C01786=1124.432,191.040,-64.237,-179.146,9.228,149.571
C01787=1124.436,190.791,-64.212,-179.148,9.226,149.571
C01788=1124.441,190.542,-64.188,-179.151,9.223,149.571
C01789=1124.446,190.294,-64.164,-179.153,9.220,149.570
C01790=1124.450,190.046,-64.139,-179.155,9.217,149.570
C01791=1124.455,189.796,-64.114,-179.157,9.214,149.570
C01792=1124.459,189.548,-64.090,-179.159,9.211,149.570
C01793=1124.464,189.299,-64.067,-179.161,9.209,149.570
C01794=1124.469,189.050,-64.042,-179.164,9.206,149.570
C01795=1124.473,188.801,-64.018,-179.166,9.204,149.570
C01796=1124.477,188.553,-63.994,-179.168,9.200,149.570
C01797=1124.482,188.304,-63.969,-179.170,9.198,149.570
C01798=1124.487,188.055,-63.946,-179.172,9.195,149.570
C01799=1124.491,187.806,-63.922,-179.175,9.192,149.570
C01800=1124.495,187.557,-63.897,-179.177,9.190,149.570
C01801=1124.500,187.309,-63.873,-179.179,9.186,149.570
C01802=1124.505,187.059,-63.849,-179.182,9.184,149.570
C01803=1124.509,186.811,-63.825,-179.184,9.181,149.570
C01804=1124.514,186.563,-63.801,-179.187,9.178,149.570
C01805=1124.519,186.313,-63.777,-179.189,9.175,149.570
C01806=1124.523,186.064,-63.753,-179.192,9.172,149.570
C01807=1124.528,185.850,-63.732,-179.194,9.170,149.570
C01808=1124.530,185.637,-63.711,-179.196,9.167,149.570
C01809=1124.534,185.422,-63.691,-179.198,9.164,149.570
C01810=1124.539,185.208,-63.670,-179.200,9.162,149.570
C01811=1124.543,184.994,-63.649,-179.202,9.160,149.570
C01812=1124.547,184.780,-63.630,-179.205,9.157,149.570
C01813=1124.550,184.566,-63.608,-179.207,9.155,149.570
C01814=1124.555,184.352,-63.588,-179.209,9.151,149.570
C01815=1124.559,184.102,-63.564,-179.212,9.148,149.570
C01816=1124.563,183.854,-63.540,-179.214,9.145,149.570
C01817=1124.568,183.605,-63.517,-179.217,9.142,149.570
C01818=1124.572,183.357,-63.493,-179.220,9.139,149.570
C01819=1124.577,183.108,-63.468,-179.222,9.136,149.570
C01820=1124.581,182.859,-63.445,-179.225,9.133,149.570
C01821=1124.586,182.611,-63.421,-179.227,9.130,149.570
C01822=1124.591,182.361,-63.397,-179.230,9.127,149.570
C01823=1124.596,182.112,-63.374,-179.233,9.124,149.570
C01824=1124.600,181.864,-63.350,-179.236,9.120,149.570
C01825=1124.604,181.614,-63.326,-179.239,9.117,149.570
C01826=1124.609,181.366,-63.302,-179.241,9.114,149.570
C01827=1124.613,181.117,-63.279,-179.244,9.111,149.570
C01828=1124.618,180.868,-63.254,-179.247,9.107,149.570
C01829=1124.623,180.619,-63.231,-179.250,9.104,149.570
C01830=1124.627,180.370,-63.208,-179.252,9.101,149.570
C01831=1124.632,180.122,-63.184,-179.256,9.098,149.570
C01832=1124.636,179.873,-63.160,-179.258,9.095,149.570
C01833=1124.641,179.624,-63.137,-179.261,9.091,149.570
C01834=1124.645,179.375,-63.113,-179.264,9.088,149.570
C01835=1124.650,179.126,-63.089,-179.267,9.085,149.570
C01836=1124.654,178.878,-63.067,-179.269,9.081,149.570
C01837=1124.659,178.629,-63.043,-179.271,9.079,149.570
C01838=1124.663,178.380,-63.019,-179.273,9.076,149.569
C01839=1124.668,178.131,-62.996,-179.276,9.073,149.569
C01840=1124.673,177.882,-62.973,-179.277,9.070,149.569
C01841=1124.677,177.633,-62.949,-179.280,9.067,149.569
C01842=1124.682,177.385,-62.925,-179.282,9.064,149.569
C01843=1124.686,177.136,-62.902,-179.284,9.061,149.569
C01844=1124.691,176.887,-62.878,-179.286,9.058,149.569
C01845=1124.696,176.638,-62.855,-179.288,9.055,149.569
C01846=1124.700,176.389,-62.832,-179.290,9.052,149.569
C01847=1124.704,176.140,-62.809,-179.293,9.049,149.568
C01848=1124.709,175.891,-62.785,-179.294,9.047,149.568
C01849=1124.714,175.642,-62.762,-179.297,9.043,149.568
C01850=1124.718,175.393,-62.738,-179.299,9.040,149.568
C01851=1124.723,175.144,-62.715,-179.301,9.038,149.568
C01852=1124.727,174.896,-62.692,-179.304,9.035,149.568
C01853=1124.732,174.647,-62.669,-179.306,9.031,149.568
C01854=1124.737,174.398,-62.646,-179.308,9.028,149.568
C01855=1124.742,174.149,-62.622,-179.310,9.026,149.568
C01856=1124.746,173.900,-62.599,-179.313,9.022,149.568
C01857=1124.750,173.652,-62.576,-179.315,9.019,149.567
C01858=1124.755,173.402,-62.553,-179.317,9.017,149.567
C01859=1124.760,173.153,-62.529,-179.319,9.014,149.567
C01860=1124.764,172.904,-62.506,-179.321,9.010,149.567
C01861=1124.768,172.656,-62.483,-179.324,9.007,149.567
C01862=1124.773,172.407,-62.460,-179.326,9.005,149.567
C01863=1124.778,172.193,-62.440,-179.328,9.002,149.567
C01864=1124.781,171.979,-62.420,-179.330,8.999,149.567
C01865=1124.785,171.764,-62.400,-179.331,8.997,149.567
C01866=1124.789,171.550,-62.380,-179.333,8.994,149.567
C01867=1124.793,171.336,-62.361,-179.335,8.992,149.567
C01868=1124.797,171.122,-62.341,-179.337,8.988,149.566
C01869=1124.801,170.908,-62.320,-179.339,8.986,149.566
C01870=1124.805,170.694,-62.301,-179.341,8.984,149.566
C01871=1124.810,170.445,-62.278,-179.344,8.981,149.566
C01872=1124.814,170.196,-62.255,-179.346,8.977,149.566
C01873=1124.819,169.947,-62.232,-179.348,8.974,149.566
C01874=1124.823,169.698,-62.208,-179.350,8.972,149.566
C01875=1124.827,169.449,-62.186,-179.353,8.969,149.566
C01876=1124.833,169.200,-62.163,-179.355,8.965,149.566
C01877=1124.837,168.951,-62.140,-179.357,8.962,149.566
C01878=1124.841,168.703,-62.117,-179.360,8.959,149.566
C01879=1124.846,168.454,-62.094,-179.362,8.955,149.565
C01880=1124.851,168.204,-62.071,-179.364,8.953,149.565
C01881=1124.856,167.956,-62.049,-179.366,8.950,149.565
C01882=1124.860,167.707,-62.025,-179.369,8.947,149.565
C01883=1124.864,167.458,-62.003,-179.371,8.943,149.565
C01884=1124.869,167.209,-61.980,-179.373,8.940,149.565
C01885=1124.875,166.960,-61.957,-179.376,8.937,149.565
C01886=1124.879,166.712,-61.934,-179.378,8.934,149.565
C01887=1124.884,166.462,-61.912,-179.381,8.931,149.565
C01888=1124.888,166.213,-61.889,-179.383,8.927,149.565
C01889=1124.893,165.965,-61.866,-179.385,8.925,149.565
C01890=1124.897,165.715,-61.844,-179.387,8.922,149.564
C01891=1124.902,165.466,-61.820,-179.390,8.919,149.564
C01892=1124.906,165.218,-61.798,-179.392,8.915,149.564
C01893=1124.911,164.969,-61.775,-179.395,8.912,149.564
C01894=1124.915,164.720,-61.753,-179.397,8.909,149.564
C01895=1124.920,164.470,-61.730,-179.399,8.906,149.564
C01896=1124.925,164.222,-61.708,-179.402,8.903,149.564
C01897=1124.930,163.973,-61.685,-179.404,8.899,149.564
C01898=1124.934,163.724,-61.662,-179.406,8.896,149.564
C01899=1124.939,163.475,-61.639,-179.409,8.893,149.564
C01900=1124.944,163.226,-61.617,-179.411,8.889,149.563
C01901=1124.947,162.978,-61.594,-179.414,8.886,149.563
C01902=1124.952,162.728,-61.572,-179.416,8.883,149.563
C01903=1124.957,162.480,-61.549,-179.419,8.880,149.563
C01904=1124.962,162.230,-61.527,-179.421,8.877,149.563
C01905=1124.966,161.981,-61.505,-179.423,8.873,149.563
C01906=1124.971,161.733,-61.482,-179.426,8.870,149.563
C01907=1124.976,161.483,-61.460,-179.428,8.867,149.563
C01908=1124.980,161.235,-61.437,-179.430,8.864,149.563
C01909=1124.985,160.986,-61.415,-179.433,8.861,149.563
C01910=1124.989,160.737,-61.392,-179.435,8.857,149.563
C01911=1124.994,160.488,-61.370,-179.438,8.853,149.563
C01912=1124.999,160.239,-61.348,-179.441,8.850,149.562
C01913=1125.003,159.990,-61.325,-179.443,8.847,149.562
C01914=1125.008,159.741,-61.303,-179.445,8.844,149.562
C01915=1125.012,159.492,-61.281,-179.447,8.840,149.562
C01916=1125.017,159.243,-61.258,-179.450,8.837,149.562
C01917=1125.022,158.994,-61.236,-179.452,8.834,149.562
C01918=1125.026,158.745,-61.214,-179.454,8.830,149.562
C01919=1125.030,158.531,-61.195,-179.457,8.827,149.562
C01920=1125.034,158.316,-61.176,-179.459,8.824,149.562
C01921=1125.038,158.102,-61.157,-179.461,8.821,149.561
C01922=1125.043,157.888,-61.138,-179.463,8.818,149.561
C01923=1125.047,157.674,-61.118,-179.465,8.816,149.561
C01924=1125.050,157.459,-61.099,-179.467,8.813,149.561
C01925=1125.054,157.245,-61.080,-179.470,8.809,149.561
C01926=1125.058,157.031,-61.061,-179.471,8.807,149.561
C01927=1125.063,156.782,-61.039,-179.474,8.804,149.561
C01928=1125.068,156.532,-61.017,-179.477,8.800,149.561
C01929=1125.073,156.284,-60.994,-179.479,8.796,149.561
C01930=1125.077,156.035,-60.972,-179.482,8.793,149.561
C01931=1125.082,155.786,-60.950,-179.484,8.790,149.560
C01932=1125.086,155.537,-60.928,-179.487,8.786,149.560
C01933=1125.090,155.288,-60.906,-179.489,8.782,149.560
C01934=1125.096,155.039,-60.884,-179.491,8.779,149.560
C01935=1125.101,154.790,-60.862,-179.494,8.776,149.560
C01936=1125.105,154.541,-60.840,-179.497,8.772,149.560
C01937=1125.110,154.292,-60.819,-179.499,8.768,149.559
C01938=1125.114,154.043,-60.797,-179.501,8.765,149.559
C01939=1125.119,153.794,-60.775,-179.504,8.761,149.559
C01940=1125.123,153.545,-60.753,-179.507,8.758,149.559
C01941=1125.128,153.296,-60.731,-179.509,8.754,149.559
C01942=1125.133,153.047,-60.709,-179.512,8.750,149.559
C01943=1125.138,152.798,-60.687,-179.514,8.747,149.559
C01944=1125.142,152.549,-60.665,-179.516,8.744,149.559
C01945=1125.147,152.300,-60.643,-179.519,8.740,149.558
C01946=1125.152,152.051,-60.621,-179.521,8.736,149.558
C01947=1125.156,151.802,-60.599,-179.524,8.732,149.558
C01948=1125.161,151.553,-60.578,-179.526,8.729,149.558
C01949=1125.166,151.304,-60.556,-179.529,8.726,149.558
C01950=1125.170,151.055,-60.534,-179.532,8.721,149.558
C01951=1125.175,150.805,-60.513,-179.534,8.718,149.557
C01952=1125.180,150.557,-60.491,-179.537,8.714,149.557
C01953=1125.185,150.308,-60.469,-179.539,8.711,149.557
C01954=1125.189,150.059,-60.447,-179.542,8.707,149.557
C01955=1125.194,149.810,-60.426,-179.544,8.703,149.557
C01956=1125.199,149.561,-60.405,-179.547,8.699,149.557
C01957=1125.203,149.311,-60.383,-179.549,8.696,149.557
C01958=1125.208,149.063,-60.361,-179.552,8.692,149.556
C01959=1125.213,148.814,-60.339,-179.554,8.688,149.556
C01960=1125.217,148.565,-60.318,-179.557,8.684,149.556
C01961=1125.222,148.316,-60.297,-179.559,8.681,149.556
C01962=1125.227,148.067,-60.275,-179.562,8.676,149.556
C01963=1125.231,147.818,-60.253,-179.564,8.673,149.555
C01964=1125.236,147.569,-60.232,-179.567,8.669,149.555
C01965=1125.241,147.320,-60.210,-179.569,8.666,149.555
C01966=1125.246,147.070,-60.189,-179.572,8.661,149.555
C01967=1125.250,146.821,-60.167,-179.575,8.657,149.555
C01968=1125.255,146.573,-60.146,-179.577,8.654,149.554
C01969=1125.259,146.323,-60.125,-179.580,8.650,149.554
C01970=1125.264,146.074,-60.103,-179.582,8.646,149.554
C01971=1125.269,145.825,-60.082,-179.585,8.642,149.554
C01972=1125.274,145.577,-60.061,-179.588,8.638,149.554
C01973=1125.278,145.328,-60.039,-179.590,8.634,149.554
C01974=1125.283,145.078,-60.018,-179.592,8.630,149.553
C01975=1125.287,144.863,-60.000,-179.594,8.627,149.553
C01976=1125.290,144.650,-59.981,-179.595,8.624,149.553
C01977=1125.295,144.435,-59.963,-179.596,8.621,149.552
C01978=1125.299,144.220,-59.945,-179.598,8.619,149.552
C01979=1125.303,144.007,-59.926,-179.599,8.616,149.552
C01980=1125.308,143.792,-59.908,-179.600,8.613,149.552
C01981=1125.311,143.577,-59.890,-179.601,8.610,149.551
C01982=1125.315,143.363,-59.871,-179.603,8.607,149.551
C01983=1125.320,143.114,-59.851,-179.604,8.603,149.550
C01984=1125.324,142.864,-59.829,-179.606,8.600,149.550
C01985=1125.329,142.616,-59.808,-179.607,8.597,149.550
C01986=1125.334,142.367,-59.787,-179.609,8.594,149.550
C01987=1125.339,142.118,-59.766,-179.611,8.590,149.549
C01988=1125.344,141.869,-59.745,-179.612,8.587,149.549
C01989=1125.348,141.619,-59.723,-179.614,8.583,149.548
C01990=1125.352,141.371,-59.702,-179.615,8.580,149.548
C01991=1125.358,141.121,-59.681,-179.617,8.577,149.548
C01992=1125.362,140.873,-59.660,-179.618,8.574,149.547
C01993=1125.367,140.624,-59.639,-179.620,8.570,149.547
C01994=1125.371,140.374,-59.618,-179.621,8.567,149.547
C01995=1125.376,140.125,-59.597,-179.623,8.564,149.546
C01996=1125.381,139.876,-59.576,-179.624,8.561,149.546
C01997=1125.386,139.627,-59.555,-179.626,8.557,149.546
C01998=1125.390,139.378,-59.535,-179.627,8.554,149.545
C01999=1125.395,139.129,-59.513,-179.629,8.551,149.545
C02000=1125.399,138.880,-59.492,-179.630,8.547,149.545
C02001=1125.404,138.630,-59.471,-179.632,8.544,149.544
C02002=1125.409,138.381,-59.450,-179.634,8.541,149.544
C02003=1125.414,138.133,-59.429,-179.635,8.537,149.544
C02004=1125.419,137.884,-59.408,-179.637,8.535,149.544
C02005=1125.423,137.635,-59.388,-179.638,8.531,149.543
C02006=1125.428,137.385,-59.367,-179.640,8.527,149.543
C02007=1125.432,137.137,-59.346,-179.641,8.524,149.543
C02008=1125.437,136.887,-59.324,-179.643,8.521,149.542
C02009=1125.442,136.638,-59.303,-179.644,8.518,149.542
C02010=1125.447,136.389,-59.283,-179.647,8.514,149.542
C02011=1125.452,136.140,-59.262,-179.648,8.511,149.541
C02012=1125.456,135.891,-59.242,-179.650,8.508,149.541
C02013=1125.461,135.642,-59.220,-179.651,8.505,149.541
C02014=1125.466,135.393,-59.200,-179.653,8.501,149.541
C02015=1125.471,135.144,-59.179,-179.655,8.497,149.540
C02016=1125.475,134.895,-59.158,-179.656,8.495,149.540
C02017=1125.480,134.646,-59.137,-179.658,8.491,149.539
C02018=1125.485,134.397,-59.117,-179.659,8.488,149.539
C02019=1125.489,134.147,-59.096,-179.661,8.485,149.539
C02020=1125.494,133.898,-59.075,-179.662,8.482,149.539
C02021=1125.498,133.649,-59.055,-179.664,8.478,149.538
C02022=1125.503,133.400,-59.034,-179.667,8.475,149.538
C02023=1125.508,133.151,-59.014,-179.668,8.471,149.538
C02024=1125.513,132.901,-58.993,-179.670,8.468,149.537
C02025=1125.517,132.652,-58.972,-179.671,8.465,149.537
C02026=1125.523,132.403,-58.951,-179.673,8.461,149.537
C02027=1125.527,132.154,-58.931,-179.675,8.458,149.537
C02028=1125.532,131.905,-58.911,-179.676,8.455,149.536
C02029=1125.537,131.656,-58.890,-179.678,8.451,149.536
C02030=1125.541,131.407,-58.869,-179.679,8.449,149.536
C02031=1125.546,131.192,-58.851,-179.681,8.445,149.535
C02032=1125.550,130.978,-58.833,-179.683,8.442,149.535
C02033=1125.553,130.764,-58.816,-179.684,8.440,149.535
C02034=1125.557,130.549,-58.799,-179.686,8.437,149.535
C02035=1125.562,130.335,-58.781,-179.687,8.434,149.534
C02036=1125.566,130.120,-58.763,-179.688,8.431,149.534
C02037=1125.570,129.906,-58.745,-179.690,8.428,149.534
C02038=1125.574,129.691,-58.728,-179.691,8.426,149.534
C02039=1125.579,129.442,-58.707,-179.693,8.422,149.533
C02040=1125.584,129.193,-58.687,-179.695,8.419,149.533
C02041=1125.588,128.944,-58.667,-179.696,8.416,149.533
C02042=1125.593,128.695,-58.646,-179.698,8.412,149.533
C02043=1125.598,128.446,-58.625,-179.700,8.409,149.532
C02044=1125.603,128.196,-58.606,-179.702,8.406,149.532
C02045=1125.608,127.947,-58.585,-179.703,8.402,149.532
C02046=1125.612,127.698,-58.564,-179.705,8.399,149.531
C02047=1125.617,127.449,-58.544,-179.707,8.396,149.531
C02048=1125.621,127.200,-58.524,-179.709,8.392,149.531
C02049=1125.627,126.950,-58.503,-179.711,8.389,149.531
C02050=1125.631,126.701,-58.483,-179.712,8.386,149.530
C02051=1125.635,126.452,-58.463,-179.714,8.382,149.530
C02052=1125.640,126.204,-58.442,-179.716,8.379,149.530
C02053=1125.645,125.954,-58.422,-179.717,8.376,149.529
C02054=1125.650,125.705,-58.402,-179.719,8.372,149.529
C02055=1125.655,125.456,-58.382,-179.721,8.369,149.529
C02056=1125.660,125.207,-58.362,-179.723,8.366,149.529
C02057=1125.664,124.958,-58.342,-179.724,8.362,149.528
C02058=1125.669,124.709,-58.321,-179.726,8.359,149.528
C02059=1125.674,124.459,-58.301,-179.728,8.355,149.528
C02060=1125.678,124.210,-58.281,-179.730,8.352,149.528
C02061=1125.683,123.961,-58.260,-179.732,8.349,149.527
C02062=1125.688,123.712,-58.241,-179.734,8.345,149.527
C02063=1125.693,123.463,-58.221,-179.735,8.342,149.527
C02064=1125.697,123.214,-58.201,-179.737,8.339,149.527
C02065=1125.703,122.965,-58.180,-179.739,8.335,149.526
C02066=1125.707,122.716,-58.160,-179.741,8.331,149.526
C02067=1125.712,122.466,-58.140,-179.742,8.329,149.526
C02068=1125.716,122.217,-58.119,-179.744,8.325,149.525
C02069=1125.722,121.968,-58.100,-179.746,8.322,149.525
C02070=1125.726,121.719,-58.080,-179.748,8.318,149.525
C02071=1125.731,121.470,-58.060,-179.749,8.315,149.525
C02072=1125.735,121.221,-58.040,-179.752,8.312,149.524
C02073=1125.740,120.971,-58.020,-179.754,8.308,149.524
C02074=1125.744,120.722,-58.000,-179.756,8.305,149.524
C02075=1125.750,120.473,-57.980,-179.757,8.302,149.524
C02076=1125.755,120.224,-57.960,-179.759,8.298,149.523
C02077=1125.760,119.975,-57.940,-179.761,8.295,149.523
C02078=1125.764,119.726,-57.919,-179.763,8.291,149.523
C02079=1125.769,119.476,-57.900,-179.765,8.288,149.523
C02080=1125.774,119.227,-57.881,-179.766,8.285,149.522
C02081=1125.779,118.978,-57.860,-179.768,8.281,149.522
C02082=1125.783,118.729,-57.841,-179.770,8.277,149.522
C02083=1125.788,118.480,-57.820,-179.772,8.274,149.522
C02084=1125.793,118.231,-57.801,-179.774,8.270,149.521
C02085=1125.798,117.981,-57.781,-179.776,8.268,149.521
C02086=1125.802,117.732,-57.761,-179.777,8.264,149.521
C02087=1125.807,117.518,-57.744,-179.779,8.260,149.520
C02088=1125.810,117.303,-57.728,-179.781,8.258,149.520
C02089=1125.815,117.089,-57.711,-179.782,8.255,149.520
C02090=1125.818,116.874,-57.693,-179.784,8.251,149.520
C02091=1125.823,116.660,-57.677,-179.786,8.249,149.520
C02092=1125.827,116.445,-57.659,-179.787,8.246,149.519
C02093=1125.831,116.230,-57.643,-179.789,8.243,149.519
C02094=1125.835,116.016,-57.625,-179.791,8.240,149.519
C02095=1125.840,115.766,-57.605,-179.793,8.236,149.519
C02096=1125.845,115.517,-57.586,-179.795,8.233,149.518
C02097=1125.850,115.268,-57.566,-179.796,8.230,149.518
C02098=1125.855,115.018,-57.547,-179.798,8.226,149.518
C02099=1125.859,114.770,-57.527,-179.800,8.223,149.518
C02100=1125.864,114.521,-57.508,-179.802,8.219,149.517
C02101=1125.868,114.271,-57.488,-179.804,8.216,149.517
C02102=1125.874,114.022,-57.469,-179.806,8.212,149.517
C02103=1125.878,113.773,-57.449,-179.808,8.208,149.516
C02104=1125.883,113.523,-57.429,-179.810,8.205,149.516
C02105=1125.888,113.275,-57.409,-179.812,8.201,149.516
C02106=1125.892,113.026,-57.390,-179.813,8.198,149.516
C02107=1125.897,112.776,-57.371,-179.815,8.195,149.515
C02108=1125.902,112.527,-57.351,-179.817,8.191,149.515
C02109=1125.907,112.278,-57.332,-179.819,8.188,149.515
C02110=1125.912,112.029,-57.312,-179.821,8.184,149.515
C02111=1125.917,111.779,-57.293,-179.823,8.180,149.514
C02112=1125.921,111.530,-57.274,-179.825,8.177,149.514
C02113=1125.926,111.281,-57.254,-179.827,8.173,149.514
C02114=1125.931,111.031,-57.235,-179.829,8.170,149.514
C02115=1125.937,110.783,-57.215,-179.831,8.166,149.513
C02116=1125.941,110.533,-57.196,-179.834,8.162,149.513
C02117=1125.945,110.284,-57.177,-179.836,8.159,149.513
C02118=1125.951,110.035,-57.157,-179.838,8.154,149.513
C02119=1125.955,109.785,-57.138,-179.840,8.151,149.512
C02120=1125.960,109.537,-57.119,-179.843,8.147,149.512
C02121=1125.965,109.287,-57.099,-179.846,8.142,149.512
C02122=1125.969,109.038,-57.080,-179.848,8.139,149.512
C02123=1125.974,108.789,-57.061,-179.850,8.134,149.512
C02124=1125.979,108.539,-57.041,-179.853,8.131,149.511
C02125=1125.984,108.291,-57.022,-179.855,8.127,149.511
C02126=1125.988,108.041,-57.003,-179.857,8.123,149.511
C02127=1125.994,107.792,-56.985,-179.860,8.119,149.511
C02128=1125.999,107.542,-56.965,-179.862,8.115,149.511
C02129=1126.003,107.294,-56.946,-179.865,8.111,149.510
C02130=1126.008,107.044,-56.927,-179.867,8.108,149.510
C02131=1126.013,106.796,-56.908,-179.869,8.103,149.510
C02132=1126.018,106.545,-56.889,-179.871,8.099,149.509
C02133=1126.023,106.297,-56.870,-179.874,8.095,149.509
C02134=1126.027,106.047,-56.851,-179.876,8.092,149.509
C02135=1126.032,105.798,-56.831,-179.878,8.088,149.509
C02136=1126.037,105.549,-56.813,-179.880,8.083,149.508
C02137=1126.042,105.300,-56.794,-179.882,8.080,149.508
C02138=1126.046,105.050,-56.775,-179.885,8.076,149.508
C02139=1126.051,104.802,-56.755,-179.887,8.072,149.508
C02140=1126.056,104.552,-56.737,-179.889,8.068,149.507
C02141=1126.061,104.303,-56.718,-179.891,8.064,149.507
C02142=1126.066,104.054,-56.699,-179.893,8.061,149.507
C02143=1126.070,103.839,-56.683,-179.895,8.057,149.506
C02144=1126.074,103.624,-56.666,-179.897,8.053,149.506
C02145=1126.078,103.410,-56.650,-179.899,8.050,149.506
C02146=1126.082,103.194,-56.633,-179.900,8.047,149.506
C02147=1126.086,102.980,-56.617,-179.902,8.043,149.505
C02148=1126.091,102.765,-56.601,-179.904,8.040,149.505
C02149=1126.095,102.551,-56.585,-179.906,8.036,149.505
C02150=1126.099,102.335,-56.569,-179.908,8.033,149.505
C02151=1126.104,102.087,-56.550,-179.910,8.029,149.504
C02152=1126.108,101.838,-56.532,-179.912,8.025,149.504
C02153=1126.113,101.588,-56.513,-179.913,8.021,149.504
C02154=1126.118,101.339,-56.494,-179.916,8.017,149.503
C02155=1126.124,101.090,-56.475,-179.918,8.013,149.503
C02156=1126.128,100.841,-56.456,-179.920,8.010,149.503
C02157=1126.133,100.591,-56.438,-179.922,8.005,149.502
C02158=1126.137,100.342,-56.419,-179.924,8.001,149.502
C02159=1126.142,100.093,-56.401,-179.926,7.998,149.502
C02160=1126.148,99.843,-56.382,-179.928,7.994,149.501
C02161=1126.152,99.594,-56.363,-179.930,7.989,149.501
C02162=1126.157,99.345,-56.345,-179.932,7.985,149.501
C02163=1126.162,99.096,-56.326,-179.934,7.982,149.500
C02164=1126.167,98.846,-56.307,-179.935,7.978,149.500
C02165=1126.171,98.597,-56.289,-179.937,7.973,149.499
C02166=1126.177,98.348,-56.270,-179.940,7.970,149.499
C02167=1126.182,98.099,-56.252,-179.941,7.966,149.499
C02168=1126.186,97.849,-56.234,-179.943,7.962,149.498
C02169=1126.191,97.600,-56.215,-179.945,7.957,149.498
C02170=1126.196,97.351,-56.197,-179.947,7.954,149.498
C02171=1126.201,97.101,-56.178,-179.949,7.950,149.497
C02172=1126.205,96.853,-56.159,-179.950,7.946,149.497
C02173=1126.211,96.603,-56.141,-179.952,7.942,149.496
C02174=1126.216,96.354,-56.123,-179.953,7.938,149.496
C02175=1126.220,96.104,-56.105,-179.956,7.934,149.496
C02176=1126.225,95.855,-56.086,-179.958,7.930,149.495
C02177=1126.230,95.606,-56.068,-179.959,7.926,149.495
C02178=1126.235,95.357,-56.049,-179.961,7.922,149.495
C02179=1126.240,95.107,-56.031,-179.962,7.919,149.494
C02180=1126.244,94.858,-56.013,-179.964,7.915,149.494
C02181=1126.249,94.609,-55.994,-179.966,7.911,149.493
C02182=1126.254,94.360,-55.976,-179.967,7.907,149.493
C02183=1126.259,94.110,-55.957,-179.969,7.903,149.492
C02184=1126.264,93.861,-55.939,-179.972,7.899,149.492
C02185=1126.269,93.611,-55.921,-179.973,7.895,149.492
C02186=1126.274,93.362,-55.903,-179.975,7.891,149.491
C02187=1126.279,93.113,-55.885,-179.976,7.887,149.491
C02188=1126.283,92.864,-55.866,-179.978,7.883,149.490
C02189=1126.288,92.615,-55.848,-179.980,7.879,149.490
C02190=1126.293,92.365,-55.830,-179.981,7.875,149.490
C02191=1126.298,92.116,-55.812,-179.983,7.871,149.489
C02192=1126.303,91.867,-55.794,-179.984,7.867,149.489
C02193=1126.308,91.618,-55.776,-179.985,7.863,149.488
C02194=1126.312,91.368,-55.758,-179.987,7.859,149.488
C02195=1126.317,91.119,-55.740,-179.989,7.856,149.487
C02196=1126.322,90.869,-55.722,-179.990,7.852,149.487
C02197=1126.327,90.620,-55.704,-179.992,7.848,149.486
C02198=1126.332,90.371,-55.686,-179.993,7.844,149.486
C02199=1126.336,90.156,-55.670,-179.994,7.841,149.486
C02200=1126.341,89.941,-55.654,-179.996,7.837,149.485
C02201=1126.345,89.727,-55.639,-179.997,7.834,149.485
C02202=1126.349,89.512,-55.623,-179.998,7.831,149.484
C02203=1126.353,89.297,-55.608,180.000,7.827,149.484
C02204=1126.357,89.082,-55.593,179.999,7.824,149.484
C02205=1126.361,88.867,-55.577,179.998,7.821,149.483
C02206=1126.365,88.652,-55.562,179.996,7.817,149.483
C02207=1126.370,88.403,-55.544,179.995,7.813,149.482
C02208=1126.375,88.154,-55.526,179.994,7.810,149.482
C02209=1126.380,87.905,-55.508,179.993,7.806,149.481
C02210=1126.385,87.656,-55.490,179.991,7.802,149.481
C02211=1126.390,87.406,-55.472,179.990,7.798,149.480
C02212=1126.395,87.157,-55.454,179.988,7.794,149.480
C02213=1126.400,86.907,-55.436,179.987,7.790,149.479
C02214=1126.405,86.658,-55.418,179.985,7.786,149.479
C02215=1126.410,86.409,-55.400,179.984,7.783,149.478
C02216=1126.415,86.159,-55.383,179.983,7.779,149.478
C02217=1126.420,85.910,-55.365,179.982,7.775,149.477
C02218=1126.425,85.661,-55.347,179.980,7.771,149.477
C02219=1126.430,85.412,-55.329,179.979,7.768,149.477
C02220=1126.434,85.162,-55.311,179.978,7.763,149.476
C02221=1126.439,84.912,-55.294,179.976,7.759,149.475
C02222=1126.443,84.663,-55.276,179.975,7.755,149.475
C02223=1126.448,84.414,-55.258,179.974,7.752,149.474
C02224=1126.453,84.164,-55.241,179.973,7.748,149.474
C02225=1126.458,83.915,-55.223,179.971,7.744,149.473
C02226=1126.463,83.666,-55.205,179.970,7.740,149.473
C02227=1126.468,83.417,-55.187,179.969,7.737,149.472
C02228=1126.473,83.167,-55.170,179.968,7.732,149.472
C02229=1126.478,82.918,-55.152,179.966,7.729,149.471
C02230=1126.482,82.669,-55.134,179.966,7.725,149.471
C02231=1126.488,82.419,-55.117,179.964,7.721,149.470
C02232=1126.493,82.170,-55.099,179.962,7.717,149.470
C02233=1126.497,81.921,-55.081,179.962,7.714,149.469
C02234=1126.502,81.671,-55.065,179.960,7.710,149.469
C02235=1126.507,81.422,-55.047,179.960,7.706,149.468
C02236=1126.512,81.172,-55.029,179.958,7.703,149.468
C02237=1126.518,80.924,-55.012,179.957,7.698,149.467
C02238=1126.523,80.674,-54.994,179.956,7.695,149.467
C02239=1126.527,80.425,-54.977,179.955,7.691,149.466
C02240=1126.532,80.176,-54.959,179.954,7.688,149.466
C02241=1126.537,79.926,-54.942,179.953,7.683,149.465
C02242=1126.542,79.677,-54.924,179.952,7.680,149.465
C02243=1126.546,79.427,-54.907,179.951,7.676,149.464
C02244=1126.551,79.178,-54.889,179.950,7.673,149.464
C02245=1126.557,78.929,-54.872,179.949,7.669,149.463
C02246=1126.562,78.679,-54.854,179.948,7.666,149.462
C02247=1126.566,78.430,-54.837,179.947,7.661,149.462
C02248=1126.571,78.181,-54.819,179.946,7.658,149.461
C02249=1126.576,77.931,-54.802,179.945,7.654,149.461
C02250=1126.580,77.682,-54.785,179.944,7.650,149.460
C02251=1126.586,77.433,-54.768,179.943,7.646,149.460
C02252=1126.591,77.184,-54.750,179.942,7.643,149.459
C02253=1126.596,76.934,-54.733,179.940,7.639,149.459
C02254=1126.601,76.684,-54.716,179.940,7.636,149.458
C02255=1126.605,76.470,-54.700,179.938,7.632,149.458
C02256=1126.609,76.255,-54.685,179.937,7.629,149.457
C02257=1126.613,76.040,-54.670,179.936,7.625,149.457
C02258=1126.618,75.825,-54.655,179.935,7.621,149.456
C02259=1126.621,75.610,-54.641,179.934,7.618,149.456
C02260=1126.626,75.396,-54.626,179.932,7.614,149.455
C02261=1126.630,75.181,-54.611,179.931,7.611,149.455
C02262=1126.635,74.966,-54.596,179.930,7.609,149.455
C02263=1126.639,74.716,-54.579,179.929,7.604,149.454
C02264=1126.644,74.467,-54.562,179.927,7.600,149.454
C02265=1126.649,74.217,-54.544,179.926,7.597,149.453
C02266=1126.654,73.969,-54.528,179.924,7.593,149.453
C02267=1126.659,73.719,-54.510,179.923,7.588,149.452
C02268=1126.664,73.469,-54.494,179.921,7.584,149.452
C02269=1126.669,73.220,-54.476,179.920,7.581,149.451
C02270=1126.674,72.970,-54.458,179.918,7.577,149.451
C02271=1126.679,72.721,-54.442,179.917,7.572,149.450
C02272=1126.684,72.472,-54.425,179.916,7.568,149.450
C02273=1126.689,72.223,-54.408,179.914,7.565,149.449
C02274=1126.694,71.973,-54.390,179.912,7.561,149.449
C02275=1126.698,71.724,-54.374,179.911,7.556,149.448
C02276=1126.703,71.474,-54.356,179.910,7.552,149.448
C02277=1126.708,71.226,-54.339,179.908,7.549,149.447
C02278=1126.713,70.976,-54.322,179.907,7.545,149.447
C02279=1126.718,70.726,-54.305,179.905,7.540,149.446
C02280=1126.723,70.477,-54.288,179.904,7.536,149.446
C02281=1126.728,70.228,-54.272,179.902,7.533,149.446
C02282=1126.733,69.978,-54.255,179.901,7.528,149.445
C02283=1126.738,69.728,-54.238,179.900,7.524,149.444
C02284=1126.743,69.479,-54.220,179.898,7.520,149.444
C02285=1126.748,69.231,-54.204,179.896,7.517,149.444
C02286=1126.752,68.981,-54.187,179.895,7.512,149.443
C02287=1126.758,68.731,-54.170,179.894,7.508,149.443
C02288=1126.762,68.482,-54.153,179.892,7.504,149.442
C02289=1126.768,68.233,-54.136,179.891,7.500,149.441
C02290=1126.772,67.983,-54.119,179.890,7.496,149.441
C02291=1126.778,67.733,-54.102,179.889,7.493,149.441
C02292=1126.783,67.485,-54.086,179.887,7.489,149.440
C02293=1126.787,67.235,-54.069,179.886,7.485,149.440
C02294=1126.792,66.985,-54.052,179.884,7.481,149.439
C02295=1126.797,66.736,-54.035,179.883,7.477,149.439
C02296=1126.802,66.487,-54.019,179.882,7.473,149.438
C02297=1126.807,66.237,-54.002,179.880,7.469,149.438
C02298=1126.812,65.988,-53.985,179.878,7.465,149.437
C02299=1126.817,65.739,-53.969,179.877,7.461,149.437
C02300=1126.822,65.489,-53.951,179.876,7.457,149.436
C02301=1126.826,65.240,-53.935,179.874,7.453,149.436
C02302=1126.832,64.991,-53.918,179.873,7.449,149.435
C02303=1126.837,64.741,-53.901,179.872,7.445,149.435
C02304=1126.842,64.491,-53.885,179.870,7.441,149.434
C02305=1126.847,64.242,-53.869,179.868,7.437,149.434
C02306=1126.852,63.992,-53.852,179.867,7.433,149.433
C02307=1126.857,63.744,-53.835,179.866,7.429,149.433
C02308=1126.861,63.494,-53.819,179.864,7.425,149.432
C02309=1126.866,63.245,-53.802,179.863,7.421,149.432
C02310=1126.872,62.996,-53.785,179.862,7.417,149.431
C02311=1126.875,62.781,-53.771,179.861,7.413,149.431
C02312=1126.880,62.565,-53.756,179.859,7.410,149.430
C02313=1126.884,62.351,-53.743,179.858,7.406,149.430
C02314=1126.889,62.135,-53.729,179.857,7.403,149.429
C02315=1126.893,61.920,-53.715,179.856,7.399,149.429
C02316=1126.898,61.705,-53.700,179.855,7.396,149.429
C02317=1126.901,61.490,-53.686,179.853,7.392,149.428
C02318=1126.906,61.275,-53.672,179.852,7.389,149.428
C02319=1126.911,61.026,-53.655,179.851,7.385,149.427
C02320=1126.915,60.777,-53.639,179.849,7.381,149.427
C02321=1126.921,60.527,-53.623,179.848,7.377,149.426
C02322=1126.925,60.278,-53.606,179.847,7.373,149.426
C02323=1126.930,60.028,-53.589,179.845,7.369,149.425
C02324=1126.935,59.779,-53.573,179.844,7.365,149.425
C02325=1126.940,59.529,-53.557,179.843,7.361,149.424
C02326=1126.945,59.280,-53.541,179.841,7.357,149.424
C02327=1126.950,59.031,-53.524,179.840,7.353,149.423
C02328=1126.955,58.781,-53.508,179.838,7.349,149.423
C02329=1126.960,58.532,-53.492,179.837,7.344,149.422
C02330=1126.965,58.282,-53.476,179.836,7.340,149.422
C02331=1126.970,58.033,-53.459,179.834,7.336,149.421
C02332=1126.975,57.784,-53.442,179.833,7.332,149.420
C02333=1126.980,57.534,-53.427,179.831,7.328,149.420
C02334=1126.985,57.285,-53.410,179.830,7.324,149.419
C02335=1126.990,57.035,-53.394,179.829,7.320,149.419
C02336=1126.995,56.786,-53.378,179.827,7.316,149.419
C02337=1127.000,56.536,-53.362,179.827,7.313,149.418
C02338=1127.005,56.287,-53.346,179.825,7.309,149.418
C02339=1127.009,56.038,-53.329,179.824,7.304,149.417
C02340=1127.015,55.788,-53.313,179.823,7.301,149.416
C02341=1127.019,55.539,-53.297,179.821,7.296,149.416
C02342=1127.025,55.289,-53.281,179.820,7.292,149.415
C02343=1127.029,55.039,-53.265,179.818,7.288,149.415
C02344=1127.035,54.791,-53.249,179.817,7.284,149.414
C02345=1127.040,54.541,-53.233,179.816,7.280,149.414
C02346=1127.044,54.292,-53.217,179.815,7.276,149.413
C02347=1127.050,54.042,-53.201,179.813,7.272,149.413
C02348=1127.054,53.793,-53.184,179.812,7.268,149.412
C02349=1127.060,53.543,-53.169,179.810,7.264,149.412
C02350=1127.064,53.294,-53.152,179.809,7.259,149.411
C02351=1127.070,53.045,-53.137,179.808,7.256,149.411
C02352=1127.075,52.795,-53.121,179.807,7.251,149.410
C02353=1127.079,52.546,-53.104,179.805,7.247,149.410
C02354=1127.085,52.296,-53.089,179.804,7.243,149.409
C02355=1127.090,52.046,-53.073,179.802,7.239,149.409
C02356=1127.095,51.797,-53.056,179.801,7.235,149.408
C02357=1127.100,51.548,-53.041,179.800,7.231,149.407
C02358=1127.105,51.298,-53.025,179.799,7.227,149.407
C02359=1127.110,51.049,-53.009,179.797,7.223,149.406
C02360=1127.115,50.800,-52.993,179.796,7.218,149.406
C02361=1127.119,50.550,-52.978,179.794,7.214,149.405
C02362=1127.124,50.301,-52.961,179.793,7.210,149.405
C02363=1127.129,50.051,-52.945,179.792,7.206,149.404
C02364=1127.135,49.802,-52.930,179.791,7.202,149.404
C02365=1127.140,49.552,-52.914,179.789,7.198,149.403
C02366=1127.144,49.303,-52.898,179.788,7.194,149.403
C02367=1127.149,49.088,-52.885,179.787,7.191,149.402
C02368=1127.153,48.872,-52.871,179.786,7.187,149.402
C02369=1127.157,48.658,-52.858,179.785,7.184,149.401
C02370=1127.161,48.442,-52.844,179.784,7.179,149.401
C02371=1127.166,48.227,-52.830,179.783,7.176,149.400
C02372=1127.170,48.012,-52.817,179.782,7.173,149.400
C02373=1127.175,47.797,-52.804,179.780,7.169,149.399
C02374=1127.179,47.582,-52.790,179.779,7.166,149.399
C02375=1127.184,47.332,-52.774,179.778,7.162,149.398
C02376=1127.189,47.083,-52.758,179.777,7.157,149.398
C02377=1127.194,46.834,-52.743,179.776,7.153,149.397
C02378=1127.199,46.584,-52.727,179.774,7.149,149.397
C02379=1127.204,46.335,-52.711,179.773,7.145,149.396
C02380=1127.209,46.086,-52.695,179.772,7.141,149.395
C02381=1127.214,45.837,-52.680,179.770,7.137,149.395
C02382=1127.219,45.586,-52.664,179.769,7.133,149.394
C02383=1127.224,45.337,-52.649,179.768,7.128,149.394
C02384=1127.230,45.088,-52.633,179.767,7.124,149.393
C02385=1127.234,44.838,-52.618,179.766,7.120,149.393
C02386=1127.239,44.588,-52.602,179.764,7.116,149.392
C02387=1127.244,44.339,-52.587,179.763,7.112,149.392
C02388=1127.249,44.090,-52.572,179.762,7.108,149.391
C02389=1127.254,43.840,-52.556,179.760,7.104,149.391
C02390=1127.259,43.590,-52.540,179.759,7.099,149.390
C02391=1127.264,43.341,-52.525,179.758,7.095,149.389
C02392=1127.269,43.092,-52.510,179.757,7.091,149.389
C02393=1127.275,42.843,-52.494,179.755,7.087,149.388
C02394=1127.279,42.593,-52.479,179.754,7.083,149.387
C02395=1127.284,42.343,-52.463,179.753,7.079,149.387
C02396=1127.289,42.094,-52.448,179.752,7.074,149.386
C02397=1127.294,41.845,-52.433,179.751,7.070,149.386
C02398=1127.300,41.595,-52.418,179.749,7.066,149.385
C02399=1127.304,41.345,-52.402,179.748,7.062,149.385
C02400=1127.309,41.096,-52.387,179.747,7.058,149.384
C02401=1127.315,40.846,-52.371,179.746,7.053,149.383
C02402=1127.319,40.597,-52.356,179.744,7.049,149.383
C02403=1127.325,40.348,-52.341,179.743,7.045,149.382
C02404=1127.329,40.099,-52.326,179.742,7.041,149.382
C02405=1127.334,39.848,-52.310,179.741,7.037,149.381
C02406=1127.339,39.599,-52.295,179.740,7.032,149.381
C02407=1127.344,39.349,-52.280,179.738,7.027,149.380
C02408=1127.350,39.100,-52.264,179.737,7.023,149.379
C02409=1127.354,38.851,-52.249,179.735,7.019,149.379
C02410=1127.360,38.601,-52.234,179.734,7.015,149.378
C02411=1127.365,38.352,-52.219,179.733,7.010,149.378
C02412=1127.370,38.102,-52.204,179.732,7.006,149.377
C02413=1127.374,37.853,-52.188,179.731,7.002,149.377
C02414=1127.380,37.603,-52.173,179.730,6.998,149.376
C02415=1127.385,37.353,-52.159,179.728,6.994,149.375
C02416=1127.390,37.104,-52.143,179.727,6.989,149.375
C02417=1127.395,36.854,-52.129,179.726,6.985,149.374
C02418=1127.400,36.605,-52.113,179.725,6.981,149.374
C02419=1127.405,36.356,-52.098,179.724,6.977,149.373
C02420=1127.411,36.106,-52.083,179.723,6.972,149.372
C02421=1127.415,35.857,-52.068,179.722,6.968,149.372
C02422=1127.420,35.608,-52.053,179.721,6.964,149.371
C02423=1127.424,35.392,-52.040,179.720,6.961,149.371
C02424=1127.429,35.176,-52.028,179.718,6.957,149.370
C02425=1127.433,34.961,-52.015,179.718,6.953,149.369
C02426=1127.438,34.747,-52.002,179.716,6.949,149.369
C02427=1127.442,34.531,-51.988,179.716,6.946,149.368
C02428=1127.447,34.316,-51.975,179.714,6.942,149.368
C02429=1127.451,34.101,-51.963,179.714,6.938,149.367
C02430=1127.455,33.886,-51.950,179.712,6.934,149.367
C02431=1127.461,33.636,-51.935,179.711,6.930,149.366
C02432=1127.465,33.387,-51.920,179.710,6.926,149.366
C02433=1127.470,33.137,-51.906,179.709,6.922,149.365
C02434=1127.475,32.887,-51.890,179.708,6.917,149.364
C02435=1127.480,32.638,-51.875,179.707,6.913,149.364
C02436=1127.485,32.389,-51.860,179.706,6.909,149.363
C02437=1127.491,32.139,-51.846,179.704,6.905,149.363
C02438=1127.495,31.889,-51.831,179.703,6.900,149.362
C02439=1127.501,31.640,-51.817,179.702,6.896,149.361
C02440=1127.506,31.391,-51.801,179.701,6.892,149.361
C02441=1127.511,31.141,-51.787,179.699,6.887,149.360
C02442=1127.516,30.892,-51.772,179.698,6.882,149.359
C02443=1127.521,30.642,-51.757,179.697,6.878,149.359
C02444=1127.526,30.393,-51.742,179.696,6.874,149.358
C02445=1127.531,30.143,-51.728,179.695,6.869,149.357
C02446=1127.536,29.894,-51.713,179.694,6.865,149.357
C02447=1127.541,29.644,-51.698,179.693,6.861,149.356
C02448=1127.546,29.395,-51.684,179.692,6.856,149.355
C02449=1127.551,29.145,-51.669,179.691,6.852,149.355
C02450=1127.556,28.896,-51.654,179.690,6.848,149.354
C02451=1127.562,28.646,-51.639,179.689,6.843,149.353
C02452=1127.567,28.396,-51.625,179.688,6.839,149.353
C02453=1127.571,28.147,-51.610,179.687,6.835,149.352
C02454=1127.576,27.897,-51.596,179.686,6.830,149.352
C02455=1127.581,27.648,-51.582,179.684,6.825,149.351
C02456=1127.587,27.398,-51.566,179.683,6.821,149.350
C02457=1127.592,27.149,-51.552,179.682,6.817,149.350
C02458=1127.597,26.899,-51.538,179.681,6.812,149.349
C02459=1127.602,26.650,-51.524,179.680,6.808,149.348
C02460=1127.607,26.401,-51.509,179.679,6.804,149.348
C02461=1127.612,26.151,-51.494,179.678,6.799,149.347
C02462=1127.617,25.901,-51.479,179.677,6.795,149.346
C02463=1127.622,25.651,-51.465,179.675,6.791,149.346
C02464=1127.627,25.402,-51.450,179.674,6.787,149.345
C02465=1127.632,25.153,-51.436,179.673,6.781,149.344
C02466=1127.637,24.903,-51.422,179.672,6.777,149.344
C02467=1127.642,24.654,-51.408,179.671,6.772,149.343
C02468=1127.647,24.404,-51.393,179.670,6.768,149.342
C02469=1127.653,24.154,-51.379,179.669,6.764,149.342
C02470=1127.658,23.905,-51.364,179.668,6.759,149.341
C02471=1127.663,23.656,-51.350,179.667,6.755,149.340
C02472=1127.668,23.406,-51.335,179.666,6.751,149.340
C02473=1127.673,23.156,-51.321,179.665,6.746,149.339
C02474=1127.678,22.907,-51.307,179.664,6.741,149.338
C02475=1127.683,22.657,-51.292,179.663,6.737,149.337
C02476=1127.688,22.407,-51.278,179.662,6.732,149.337
C02477=1127.694,22.158,-51.264,179.661,6.728,149.336
C02478=1127.698,21.909,-51.250,179.659,6.724,149.336
C02479=1127.703,21.694,-51.237,179.658,6.719,149.335
C02480=1127.707,21.478,-51.225,179.658,6.716,149.334
C02481=1127.712,21.263,-51.213,179.657,6.712,149.334
C02482=1127.716,21.048,-51.201,179.656,6.708,149.333
C02483=1127.720,20.832,-51.188,179.655,6.704,149.333
C02484=1127.725,20.617,-51.176,179.655,6.701,149.332
C02485=1127.729,20.402,-51.163,179.654,6.696,149.331
C02486=1127.733,20.186,-51.152,179.652,6.692,149.331
C02487=1127.738,19.937,-51.137,179.651,6.688,149.330
C02488=1127.744,19.688,-51.123,179.650,6.683,149.329
C02489=1127.749,19.438,-51.109,179.649,6.679,149.329
C02490=1127.754,19.188,-51.095,179.649,6.674,149.328
C02491=1127.759,18.939,-51.081,179.648,6.670,149.327
C02492=1127.764,18.690,-51.067,179.647,6.666,149.326
C02493=1127.769,18.440,-51.052,179.645,6.660,149.326
C02494=1127.774,18.189,-51.039,179.645,6.656,149.325
C02495=1127.780,17.940,-51.025,179.643,6.651,149.324
C02496=1127.784,17.691,-51.011,179.642,6.647,149.324
C02497=1127.789,17.441,-50.997,179.642,6.642,149.323
C02498=1127.795,17.192,-50.983,179.641,6.638,149.322
C02499=1127.800,16.943,-50.969,179.639,6.633,149.321
C02500=1127.805,16.693,-50.955,179.639,6.628,149.321
C02501=1127.810,16.443,-50.941,179.638,6.624,149.320
C02502=1127.815,16.194,-50.927,179.637,6.620,149.319
C02503=1127.820,15.944,-50.913,179.636,6.615,149.318
C02504=1127.825,15.694,-50.899,179.635,6.611,149.318
C02505=1127.830,15.445,-50.885,179.633,6.605,149.317
C02506=1127.835,15.195,-50.872,179.633,6.601,149.316
C02507=1127.840,14.945,-50.857,179.632,6.596,149.316
C02508=1127.846,14.696,-50.843,179.631,6.592,149.315
C02509=1127.851,14.447,-50.829,179.630,6.587,149.314
C02510=1127.856,14.197,-50.817,179.629,6.582,149.313
C02511=1127.861,13.948,-50.802,179.628,6.578,149.313
C02512=1127.866,13.698,-50.788,179.627,6.573,149.312
C02513=1127.872,13.448,-50.775,179.626,6.568,149.311
C02514=1127.876,13.199,-50.761,179.625,6.564,149.310
C02515=1127.881,12.949,-50.747,179.624,6.559,149.309
C02516=1127.887,12.700,-50.734,179.623,6.554,149.309
C02517=1127.892,12.450,-50.719,179.623,6.550,149.308
C02518=1127.897,12.201,-50.706,179.622,6.545,149.307
C02519=1127.902,11.951,-50.693,179.621,6.541,149.306
C02520=1127.907,11.701,-50.678,179.619,6.535,149.306
C02521=1127.912,11.452,-50.664,179.619,6.531,149.305
C02522=1127.917,11.202,-50.651,179.618,6.526,149.304
C02523=1127.922,10.953,-50.637,179.617,6.522,149.303
C02524=1127.928,10.703,-50.624,179.616,6.517,149.303
C02525=1127.933,10.454,-50.611,179.615,6.512,149.302
C02526=1127.938,10.204,-50.597,179.614,6.508,149.301
C02527=1127.943,9.955,-50.583,179.613,6.503,149.300
C02528=1127.948,9.705,-50.569,179.613,6.498,149.299
C02529=1127.953,9.455,-50.556,179.611,6.493,149.299
C02530=1127.958,9.206,-50.542,179.611,6.488,149.298
C02531=1127.963,8.956,-50.529,179.610,6.484,149.297
C02532=1127.968,8.707,-50.515,179.609,6.479,149.296
C02533=1127.974,8.457,-50.502,179.608,6.474,149.296
C02534=1127.979,8.208,-50.488,179.607,6.469,149.295
C02535=1127.984,7.992,-50.477,179.607,6.465,149.294
C02536=1127.988,7.776,-50.465,179.607,6.462,149.293
C02537=1127.992,7.561,-50.453,179.606,6.457,149.292
C02538=1127.996,7.346,-50.442,179.606,6.454,149.292
C02539=1128.000,7.131,-50.430,179.605,6.450,149.291
C02540=1128.005,6.915,-50.419,179.605,6.446,149.290
C02541=1128.010,6.700,-50.407,179.605,6.443,149.290
C02542=1128.015,6.485,-50.395,179.604,6.438,149.289
C02543=1128.019,6.235,-50.382,179.604,6.434,149.288
C02544=1128.025,5.986,-50.368,179.603,6.430,149.287
C02545=1128.029,5.736,-50.356,179.603,6.425,149.286
C02546=1128.035,5.486,-50.342,179.602,6.420,149.285
C02547=1128.040,5.236,-50.328,179.602,6.416,149.285
C02548=1128.045,4.987,-50.315,179.602,6.412,149.284
C02549=1128.050,4.737,-50.301,179.601,6.407,149.283
C02550=1128.055,4.488,-50.289,179.601,6.402,149.282
C02551=1128.060,4.238,-50.275,179.601,6.398,149.281
C02552=1128.065,3.989,-50.262,179.600,6.394,149.280
C02553=1128.071,3.739,-50.248,179.599,6.389,149.279
C02554=1128.076,3.489,-50.236,179.599,6.384,149.279
C02555=1128.082,3.240,-50.222,179.598,6.380,149.278
C02556=1128.086,2.990,-50.209,179.598,6.376,149.277
C02557=1128.092,2.741,-50.195,179.598,6.371,149.276
C02558=1128.096,2.491,-50.182,179.597,6.367,149.275
C02559=1128.102,2.242,-50.169,179.596,6.362,149.274
C02560=1128.107,1.992,-50.156,179.596,6.358,149.274
C02561=1128.112,1.742,-50.142,179.596,6.353,149.273
C02562=1128.117,1.493,-50.130,179.595,6.349,149.272
C02563=1128.122,1.243,-50.117,179.594,6.344,149.271
C02564=1128.127,0.994,-50.103,179.594,6.340,149.270
C02565=1128.132,0.744,-50.090,179.594,6.336,149.269
C02566=1128.138,0.494,-50.077,179.593,6.331,149.268
C02567=1128.143,0.245,-50.064,179.593,6.326,149.268
C02568=1128.149,-0.005,-50.051,179.592,6.322,149.267
C02569=1128.153,-0.254,-50.037,179.591,6.317,149.266
C02570=1128.158,-0.504,-50.025,179.591,6.312,149.265
C02571=1128.163,-0.754,-50.011,179.591,6.308,149.264
C02572=1128.168,-1.003,-49.999,179.590,6.304,149.264
C02573=1128.174,-1.253,-49.985,179.589,6.299,149.263
C02574=1128.179,-1.503,-49.972,179.589,6.295,149.262
C02575=1128.184,-1.752,-49.960,179.588,6.290,149.261
C02576=1128.190,-2.002,-49.947,179.587,6.286,149.260
C02577=1128.194,-2.251,-49.933,179.587,6.281,149.259
C02578=1128.199,-2.501,-49.920,179.587,6.277,149.259
C02579=1128.205,-2.750,-49.907,179.586,6.273,149.258
C02580=1128.209,-3.000,-49.894,179.585,6.268,149.257
C02581=1128.215,-3.250,-49.882,179.585,6.263,149.256
C02582=1128.220,-3.499,-49.868,179.584,6.258,149.255
C02583=1128.225,-3.749,-49.855,179.583,6.254,149.255
C02584=1128.230,-3.999,-49.843,179.583,6.249,149.254
C02585=1128.236,-4.248,-49.830,179.582,6.245,149.253
C02586=1128.241,-4.498,-49.817,179.581,6.240,149.252
C02587=1128.246,-4.748,-49.804,179.581,6.236,149.251
C02588=1128.251,-4.997,-49.791,179.581,6.232,149.250
C02589=1128.257,-5.247,-49.778,179.580,6.227,149.250
C02590=1128.261,-5.497,-49.765,179.579,6.223,149.249
C02591=1128.266,-5.712,-49.755,179.578,6.218,149.248
C02592=1128.270,-5.927,-49.743,179.578,6.215,149.248
C02593=1128.275,-6.143,-49.732,179.578,6.211,149.247
C02594=1128.279,-6.359,-49.721,179.577,6.206,149.246
C02595=1128.284,-6.573,-49.710,179.577,6.203,149.245
C02596=1128.288,-6.789,-49.699,179.576,6.198,149.245
C02597=1128.292,-7.005,-49.688,179.575,6.195,149.244
C02598=1128.297,-7.219,-49.677,179.575,6.191,149.243
C02599=1128.302,-7.470,-49.665,179.574,6.187,149.242
C02600=1128.308,-7.720,-49.652,179.574,6.182,149.242
C02601=1128.313,-7.969,-49.639,179.573,6.178,149.241
C02602=1128.318,-8.218,-49.626,179.572,6.173,149.240
C02603=1128.323,-8.468,-49.613,179.572,6.168,149.239
C02604=1128.328,-8.718,-49.601,179.571,6.164,149.239
C02605=1128.334,-8.967,-49.588,179.570,6.159,149.238
C02606=1128.339,-9.217,-49.576,179.570,6.154,149.237
C02607=1128.344,-9.467,-49.563,179.569,6.150,149.236
C02608=1128.349,-9.717,-49.550,179.568,6.145,149.235
C02609=1128.354,-9.966,-49.538,179.567,6.141,149.235
C02610=1128.359,-10.215,-49.525,179.567,6.136,149.234
C02611=1128.364,-10.465,-49.513,179.566,6.131,149.233
C02612=1128.370,-10.715,-49.500,179.565,6.127,149.232
C02613=1128.375,-10.965,-49.487,179.565,6.122,149.231
C02614=1128.380,-11.214,-49.474,179.564,6.118,149.230
C02615=1128.385,-11.464,-49.462,179.563,6.113,149.230
C02616=1128.390,-11.713,-49.450,179.563,6.109,149.229
C02617=1128.395,-11.963,-49.437,179.562,6.103,149.228
C02618=1128.401,-12.212,-49.425,179.561,6.099,149.227
C02619=1128.405,-12.463,-49.412,179.560,6.094,149.226
C02620=1128.411,-12.712,-49.400,179.559,6.090,149.226
C02621=1128.416,-12.961,-49.387,179.559,6.085,149.225
C02622=1128.421,-13.211,-49.375,179.558,6.080,149.224
C02623=1128.426,-13.460,-49.363,179.557,6.076,149.223
C02624=1128.432,-13.710,-49.350,179.557,6.071,149.222
C02625=1128.438,-13.960,-49.338,179.556,6.066,149.221
C02626=1128.443,-14.209,-49.325,179.555,6.062,149.221
C02627=1128.447,-14.460,-49.313,179.555,6.057,149.220
C02628=1128.453,-14.709,-49.300,179.554,6.052,149.219
C02629=1128.458,-14.959,-49.288,179.553,6.047,149.218
C02630=1128.463,-15.209,-49.276,179.552,6.043,149.218
C02631=1128.468,-15.458,-49.263,179.552,6.038,149.217
C02632=1128.474,-15.708,-49.251,179.551,6.034,149.216
C02633=1128.479,-15.957,-49.239,179.550,6.029,149.215
C02634=1128.484,-16.206,-49.226,179.550,6.024,149.214
C02635=1128.489,-16.456,-49.214,179.548,6.019,149.214
C02636=1128.494,-16.706,-49.202,179.548,6.014,149.213
C02637=1128.499,-16.955,-49.190,179.547,6.009,149.212
C02638=1128.504,-17.205,-49.178,179.546,6.005,149.211
C02639=1128.509,-17.455,-49.165,179.546,6.000,149.210
C02640=1128.514,-17.705,-49.153,179.544,5.995,149.209
C02641=1128.520,-17.955,-49.141,179.544,5.991,149.209
C02642=1128.525,-18.204,-49.129,179.543,5.986,149.208
C02643=1128.530,-18.454,-49.116,179.543,5.981,149.207
C02644=1128.536,-18.704,-49.105,179.542,5.977,149.206
C02645=1128.541,-18.953,-49.092,179.540,5.971,149.205
C02646=1128.546,-19.203,-49.080,179.540,5.966,149.204
C02647=1128.555,-19.617,-49.060,179.539,5.959,149.203
C02648=1128.564,-20.030,-49.040,179.537,5.951,149.202
C02649=1128.572,-20.444,-49.020,179.536,5.943,149.200
C02650=1128.581,-20.858,-49.000,179.535,5.935,149.199
C02651=1128.586,-21.108,-48.988,179.534,5.929,149.198
C02652=1128.591,-21.358,-48.977,179.533,5.925,149.197
C02653=1128.596,-21.607,-48.964,179.532,5.920,149.197
C02654=1128.601,-21.857,-48.952,179.532,5.915,149.196
C02655=1128.607,-22.107,-48.940,179.531,5.910,149.195
C02656=1128.612,-22.357,-48.928,179.530,5.906,149.194
C02657=1128.617,-22.606,-48.916,179.529,5.901,149.193
C02658=1128.622,-22.856,-48.904,179.528,5.895,149.192
C02659=1128.628,-23.106,-48.893,179.528,5.891,149.192
C02660=1128.633,-23.355,-48.880,179.526,5.885,149.191
C02661=1128.639,-23.605,-48.868,179.525,5.881,149.190
C02662=1128.643,-23.854,-48.857,179.525,5.876,149.189
C02663=1128.649,-24.104,-48.845,179.524,5.870,149.188
C02664=1128.654,-24.354,-48.833,179.523,5.866,149.187
C02665=1128.659,-24.603,-48.821,179.522,5.861,149.187
C02666=1128.664,-24.853,-48.809,179.521,5.856,149.186
C02667=1128.670,-25.103,-48.798,179.521,5.851,149.185
C02668=1128.675,-25.353,-48.786,179.520,5.845,149.184
C02669=1128.680,-25.603,-48.774,179.519,5.841,149.183
C02670=1128.686,-25.852,-48.763,179.518,5.836,149.182
C02671=1128.691,-26.101,-48.750,179.517,5.831,149.182
C02672=1128.696,-26.351,-48.739,179.519,5.827,149.180
C02673=1128.701,-26.601,-48.727,179.520,5.823,149.179
C02674=1128.706,-26.851,-48.715,179.522,5.820,149.178
C02675=1128.732,-28.116,-48.653,179.257,6.307,149.362
C02676=1128.741,-28.536,-48.633,179.253,6.306,149.363
C02677=1128.746,-28.785,-48.621,179.251,6.305,149.364
C02678=1128.752,-29.035,-48.610,179.248,6.304,149.364
C02679=1128.757,-29.285,-48.598,179.246,6.304,149.365
C02680=1128.762,-29.534,-48.587,179.244,6.303,149.365
C02681=1128.767,-29.784,-48.575,179.241,6.302,149.366
C02682=1128.773,-30.034,-48.563,179.239,6.302,149.366
C02683=1128.778,-30.284,-48.552,179.237,6.301,149.367
C02684=1128.783,-30.533,-48.539,179.234,6.300,149.367
C02685=1128.788,-30.783,-48.527,179.232,6.299,149.368
C02686=1128.793,-31.032,-48.516,179.229,6.298,149.368
C02687=1128.799,-31.282,-48.504,179.227,6.297,149.369
C02688=1128.804,-31.532,-48.492,179.225,6.297,149.369
C02689=1128.809,-31.781,-48.481,179.222,6.296,149.370
C02690=1128.814,-32.031,-48.469,179.220,6.295,149.371
C02691=1128.819,-32.281,-48.458,179.218,6.295,149.371
C02692=1128.825,-32.530,-48.446,179.215,6.294,149.372
C02693=1128.831,-32.780,-48.434,179.213,6.293,149.372
C02694=1128.835,-33.030,-48.423,179.210,6.293,149.373
C02695=1128.841,-33.280,-48.411,179.208,6.292,149.373
C02696=1128.845,-33.529,-48.400,179.206,6.291,149.374
C02697=1128.851,-33.779,-48.388,179.204,6.290,149.374
C02698=1128.857,-34.029,-48.377,179.201,6.290,149.375
C02699=1128.861,-34.278,-48.365,179.199,6.289,149.375
C02700=1128.867,-34.528,-48.353,179.197,6.288,149.376
C02701=1128.872,-34.778,-48.342,179.195,6.288,149.376
C02702=1128.878,-35.027,-48.331,179.192,6.287,149.377
C02703=1128.882,-35.277,-48.319,179.190,6.286,149.377
C02704=1128.888,-35.527,-48.307,179.188,6.286,149.378
C02705=1128.892,-35.776,-48.296,179.185,6.285,149.378
C02706=1128.898,-36.026,-48.284,179.183,6.284,149.379
C02707=1128.903,-36.276,-48.274,179.181,6.284,149.380
C02708=1128.909,-36.526,-48.262,179.178,6.283,149.380
C02709=1128.914,-36.775,-48.251,179.176,6.282,149.381
C02710=1128.919,-37.025,-48.239,179.174,6.282,149.381
C02711=1128.924,-37.274,-48.228,179.171,6.281,149.382
C02712=1128.930,-37.524,-48.216,179.169,6.279,149.382
C02713=1128.934,-37.774,-48.205,179.166,6.279,149.383
C02714=1128.940,-38.024,-48.193,179.164,6.278,149.383
C02715=1128.945,-38.273,-48.183,179.162,6.278,149.384
C02716=1128.951,-38.523,-48.171,179.159,6.277,149.384
C02717=1128.956,-38.773,-48.160,179.157,6.276,149.385
C02718=1128.961,-39.023,-48.148,179.155,6.276,149.385
C02719=1128.966,-39.272,-48.137,179.152,6.275,149.386
C02720=1128.972,-39.521,-48.125,179.150,6.274,149.386
C02721=1128.977,-39.772,-48.114,179.148,6.273,149.387
C02722=1128.983,-40.021,-48.103,179.145,6.273,149.388
C02723=1128.987,-40.271,-48.092,179.143,6.272,149.388
C02724=1128.993,-40.521,-48.080,179.141,6.271,149.389
C02725=1128.998,-40.770,-48.069,179.139,6.271,149.389
C02726=1129.003,-41.020,-48.058,179.136,6.270,149.390
C02727=1129.009,-41.270,-48.046,179.134,6.269,149.390
C02728=1129.013,-41.519,-48.035,179.132,6.269,149.391
C02729=1129.020,-41.769,-48.024,179.129,6.268,149.391
C02730=1129.024,-42.019,-48.013,179.127,6.267,149.392
C02731=1129.029,-42.268,-48.002,179.125,6.267,149.392
C02732=1129.035,-42.518,-47.990,179.122,6.266,149.393
C02733=1129.040,-42.768,-47.980,179.120,6.265,149.393
C02734=1129.045,-43.018,-47.968,179.119,6.265,149.394
C02735=1129.051,-43.267,-47.957,179.116,6.265,149.394
C02736=1129.056,-43.517,-47.946,179.114,6.264,149.395
C02737=1129.061,-43.767,-47.934,179.112,6.263,149.395
C02738=1129.066,-44.016,-47.923,179.109,6.262,149.396
C02739=1129.071,-44.266,-47.913,179.107,6.262,149.397
C02740=1129.077,-44.516,-47.901,179.105,6.261,149.397
C02741=1129.082,-44.765,-47.890,179.102,6.261,149.398
C02742=1129.087,-45.015,-47.879,179.100,6.260,149.398
C02743=1129.093,-45.264,-47.868,179.098,6.259,149.399
C02744=1129.098,-45.514,-47.857,179.095,6.259,149.399
C02745=1129.103,-45.764,-47.846,179.093,6.258,149.400
C02746=1129.109,-46.013,-47.834,179.091,6.257,149.400
C02747=1129.114,-46.264,-47.824,179.089,6.256,149.401
C02748=1129.119,-46.513,-47.813,179.086,6.256,149.401
C02749=1129.124,-46.762,-47.802,179.084,6.255,149.402
C02750=1129.130,-47.013,-47.790,179.082,6.254,149.402
C02751=1129.135,-47.262,-47.780,179.080,6.254,149.403
C02752=1129.140,-47.512,-47.769,179.077,6.253,149.404
C02753=1129.145,-47.762,-47.758,179.075,6.252,149.404
C02754=1129.151,-48.011,-47.747,179.072,6.252,149.404
C02755=1129.156,-48.261,-47.736,179.070,6.251,149.405
C02756=1129.161,-48.511,-47.725,179.068,6.251,149.406
C02757=1129.167,-48.761,-47.714,179.065,6.250,149.406
C02758=1129.172,-49.010,-47.703,179.063,6.249,149.407
C02759=1129.177,-49.260,-47.692,179.061,6.248,149.407
C02760=1129.182,-49.510,-47.681,179.059,6.248,149.408
C02761=1129.187,-49.759,-47.671,179.057,6.248,149.408
C02762=1129.193,-50.010,-47.659,179.055,6.247,149.409
C02763=1129.198,-50.258,-47.648,179.052,6.246,149.409
C02764=1129.203,-50.509,-47.638,179.050,6.246,149.410
C02765=1129.210,-50.779,-47.626,179.048,6.245,149.410
C02766=1129.215,-51.050,-47.614,179.045,6.244,149.411
C02767=1129.220,-51.321,-47.602,179.043,6.243,149.411
C02768=1129.227,-51.591,-47.591,179.040,6.242,149.412
C02769=1129.231,-51.841,-47.580,179.038,6.242,149.413
C02770=1129.237,-52.091,-47.569,179.036,6.242,149.413
C02771=1129.243,-52.341,-47.558,179.034,6.241,149.414
C02772=1129.247,-52.591,-47.547,179.031,6.241,149.414
C02773=1129.253,-52.840,-47.537,179.029,6.240,149.415
C02774=1129.258,-53.090,-47.525,179.027,6.239,149.415
C02775=1129.263,-53.340,-47.515,179.025,6.238,149.416
C02776=1129.268,-53.590,-47.505,179.022,6.238,149.416
C02777=1129.273,-53.839,-47.494,179.020,6.237,149.417
C02778=1129.279,-54.089,-47.483,179.018,6.236,149.417
C02779=1129.285,-54.339,-47.472,179.015,6.236,149.418
C02780=1129.289,-54.588,-47.461,179.013,6.235,149.418
C02781=1129.295,-54.838,-47.451,179.011,6.234,149.419
C02782=1129.300,-55.088,-47.440,179.009,6.235,149.419
C02783=1129.305,-55.337,-47.429,179.007,6.234,149.420
C02784=1129.310,-55.587,-47.419,179.005,6.233,149.420
C02785=1129.316,-55.837,-47.409,179.002,6.232,149.421
C02786=1129.321,-56.087,-47.397,179.000,6.232,149.422
C02787=1129.326,-56.336,-47.387,178.998,6.231,149.422
C02788=1129.331,-56.586,-47.376,178.995,6.230,149.423
C02789=1129.337,-56.835,-47.366,178.993,6.230,149.423
C02790=1129.342,-57.085,-47.355,178.991,6.229,149.424
C02791=1129.348,-57.335,-47.344,178.988,6.228,149.424
C02792=1129.353,-57.585,-47.334,178.987,6.228,149.425
C02793=1129.358,-57.835,-47.323,178.985,6.228,149.425
C02794=1129.364,-58.084,-47.312,178.982,6.227,149.426
C02795=1129.369,-58.334,-47.302,178.980,6.226,149.426
C02796=1129.374,-58.584,-47.292,178.977,6.226,149.427
C02797=1129.379,-58.834,-47.280,178.975,6.225,149.427
C02798=1129.385,-59.083,-47.270,178.973,6.224,149.428
C02799=1129.390,-59.333,-47.260,178.971,6.223,149.428
C02800=1129.395,-59.583,-47.249,178.969,6.223,149.429
C02801=1129.401,-59.832,-47.239,178.967,6.223,149.429
C02802=1129.406,-60.082,-47.228,178.964,6.222,149.430
C02803=1129.411,-60.332,-47.218,178.962,6.222,149.430
C02804=1129.416,-60.582,-47.207,178.960,6.221,149.431
C02805=1129.422,-60.831,-47.197,178.958,6.220,149.431
C02806=1129.427,-61.081,-47.187,178.956,6.219,149.432
C02807=1129.432,-61.331,-47.176,178.953,6.219,149.433
C02808=1129.438,-61.581,-47.166,178.951,6.218,149.433
C02809=1129.442,-61.830,-47.155,178.949,6.218,149.434
C02810=1129.447,-62.080,-47.145,178.947,6.217,149.434
C02811=1129.453,-62.329,-47.135,178.945,6.217,149.435
C02812=1129.458,-62.579,-47.124,178.942,6.216,149.435
C02813=1129.464,-62.829,-47.114,178.940,6.216,149.436
C02814=1129.469,-63.079,-47.103,178.938,6.215,149.436
C02815=1129.474,-63.329,-47.093,178.936,6.214,149.437
C02816=1129.480,-63.578,-47.083,178.934,6.214,149.437
C02817=1129.485,-63.828,-47.072,178.932,6.213,149.438
C02818=1129.490,-64.078,-47.062,178.929,6.213,149.438
C02819=1129.496,-64.328,-47.052,178.927,6.212,149.439
C02820=1129.501,-64.577,-47.041,178.925,6.211,149.439
C02821=1129.506,-64.827,-47.031,178.923,6.211,149.440
C02822=1129.511,-65.076,-47.021,178.920,6.210,149.440
C02823=1129.516,-65.326,-47.010,178.919,6.210,149.441
C02824=1129.522,-65.576,-47.000,178.916,6.210,149.441
C02825=1129.527,-65.825,-46.990,178.914,6.209,149.442
C02826=1129.532,-66.076,-46.979,178.912,6.208,149.442
C02827=1129.538,-66.325,-46.969,178.909,6.207,149.443
C02828=1129.544,-66.575,-46.959,178.907,6.206,149.443
C02829=1129.549,-66.825,-46.948,178.906,6.207,149.444
C02830=1129.553,-67.074,-46.939,178.903,6.206,149.445
C02831=1129.559,-67.324,-46.929,178.901,6.205,149.445
C02832=1129.564,-67.574,-46.918,178.899,6.205,149.446
C02833=1129.570,-67.824,-46.908,178.896,6.204,149.446
C02834=1129.576,-68.074,-46.898,178.894,6.203,149.447
C02835=1129.581,-68.324,-46.888,178.893,6.203,149.447
C02836=1129.585,-68.573,-46.878,178.890,6.203,149.448
C02837=1129.591,-68.823,-46.868,178.888,6.202,149.448
C02838=1129.597,-69.072,-46.858,178.886,6.201,149.449
C02839=1129.602,-69.322,-46.847,178.883,6.200,149.449
C02840=1129.607,-69.572,-46.837,178.881,6.200,149.450
C02841=1129.612,-69.821,-46.827,178.880,6.200,149.450
C02842=1129.618,-70.071,-46.817,178.877,6.199,149.451
C02843=1129.623,-70.321,-46.807,178.875,6.199,149.451
C02844=1129.629,-70.571,-46.797,178.873,6.198,149.452
C02845=1129.634,-70.821,-46.787,178.870,6.197,149.452
C02846=1129.638,-71.071,-46.777,178.869,6.197,149.453
C02847=1129.644,-71.320,-46.767,178.867,6.196,149.453
C02848=1129.650,-71.570,-46.756,178.864,6.196,149.454
C02849=1129.655,-71.819,-46.746,178.862,6.195,149.454
C02850=1129.659,-72.069,-46.736,178.860,6.195,149.455
C02851=1129.665,-72.319,-46.727,178.857,6.194,149.455
C02852=1129.671,-72.569,-46.717,178.856,6.194,149.456
C02853=1129.677,-72.818,-46.706,178.854,6.193,149.456
C02854=1129.681,-73.068,-46.697,178.851,6.192,149.457
C02855=1129.686,-73.318,-46.686,178.849,6.192,149.458
C02856=1129.692,-73.568,-46.677,178.846,6.191,149.458
C02857=1129.698,-73.818,-46.666,178.845,6.191,149.458
C02858=1129.703,-74.067,-46.657,178.843,6.190,149.459
C02859=1129.708,-74.317,-46.646,178.841,6.190,149.459
C02860=1129.714,-74.567,-46.637,178.838,6.189,149.460
C02861=1129.719,-74.816,-46.627,178.837,6.189,149.460
C02862=1129.724,-75.066,-46.617,178.834,6.189,149.461
C02863=1129.730,-75.316,-46.607,178.832,6.188,149.462
C02864=1129.735,-75.565,-46.598,178.830,6.187,149.462
C02865=1129.740,-75.816,-46.587,178.827,6.186,149.463
C02866=1129.746,-76.065,-46.577,178.826,6.186,149.463
C02867=1129.750,-76.314,-46.567,178.824,6.186,149.464
C02868=1129.756,-76.565,-46.558,178.821,6.185,149.464
C02869=1129.762,-76.836,-46.546,178.819,6.184,149.465
C02870=1129.768,-77.108,-46.536,178.817,6.184,149.465
C02871=1129.773,-77.379,-46.526,178.814,6.183,149.466
C02872=1129.780,-77.651,-46.515,178.812,6.183,149.466
C02873=1129.785,-77.900,-46.505,178.810,6.182,149.467
C02874=1129.790,-78.150,-46.496,178.808,6.182,149.467
C02875=1129.795,-78.401,-46.485,178.806,6.181,149.468
C02876=1129.800,-78.650,-46.475,178.804,6.180,149.468
C02877=1129.806,-78.900,-46.466,178.801,6.180,149.469
C02878=1129.812,-79.149,-46.456,178.800,6.180,149.469
C02879=1129.817,-79.399,-46.446,178.798,6.179,149.470
C02880=1129.823,-79.649,-46.437,178.795,6.179,149.471
C02881=1129.827,-79.898,-46.427,178.793,6.178,149.471
C02882=1129.833,-80.148,-46.418,178.791,6.178,149.471
C02883=1129.838,-80.398,-46.408,178.789,6.177,149.472
C02884=1129.843,-80.648,-46.397,178.787,6.176,149.472
C02885=1129.849,-80.898,-46.388,178.785,6.176,149.473
C02886=1129.854,-81.147,-46.378,178.783,6.176,149.473
C02887=1129.860,-81.397,-46.369,178.781,6.175,149.474
C02888=1129.865,-81.647,-46.359,178.779,6.174,149.474
C02889=1129.871,-81.897,-46.350,178.776,6.174,149.475
C02890=1129.876,-82.146,-46.340,178.774,6.174,149.476
C02891=1129.881,-82.396,-46.329,178.772,6.173,149.476
C02892=1129.886,-82.646,-46.321,178.770,6.172,149.477
C02893=1129.891,-82.896,-46.310,178.768,6.171,149.477
C02894=1129.897,-83.146,-46.301,178.766,6.172,149.478
C02895=1129.902,-83.395,-46.291,178.764,6.171,149.478
C02896=1129.908,-83.645,-46.282,178.762,6.170,149.478
C02897=1129.913,-83.894,-46.272,178.760,6.169,149.479
C02898=1129.919,-84.145,-46.263,178.757,6.170,149.480
C02899=1129.924,-84.394,-46.253,178.755,6.169,149.480
C02900=1129.929,-84.644,-46.244,178.753,6.168,149.481
C02901=1129.934,-84.893,-46.234,178.751,6.167,149.481
C02902=1129.940,-85.143,-46.225,178.749,6.167,149.482
C02903=1129.945,-85.394,-46.215,178.747,6.167,149.482
C02904=1129.950,-85.643,-46.206,178.745,6.166,149.483
C02905=1129.956,-85.893,-46.196,178.743,6.165,149.483
C02906=1129.960,-86.142,-46.186,178.741,6.165,149.484
C02907=1129.966,-86.393,-46.177,178.739,6.165,149.484
C02908=1129.971,-86.642,-46.167,178.736,6.164,149.485
C02909=1129.977,-86.892,-46.158,178.735,6.164,149.485
C02910=1129.982,-87.142,-46.149,178.732,6.163,149.486
C02911=1129.988,-87.391,-46.139,178.730,6.163,149.486
C02912=1129.993,-87.641,-46.130,178.728,6.162,149.487
C02913=1129.998,-87.891,-46.120,178.726,6.162,149.487
C02914=1130.004,-88.141,-46.111,178.724,6.161,149.488
C02915=1130.009,-88.391,-46.102,178.722,6.160,149.488
C02916=1130.015,-88.640,-46.092,178.720,6.161,149.489
C02917=1130.020,-88.890,-46.083,178.718,6.160,149.489
C02918=1130.025,-89.139,-46.073,178.716,6.159,149.490
C02919=1130.030,-89.389,-46.064,178.714,6.158,149.490
C02920=1130.036,-89.639,-46.055,178.712,6.159,149.491
C02921=1130.041,-89.889,-46.045,178.710,6.158,149.491
C02922=1130.046,-90.139,-46.036,178.707,6.157,149.492
C02923=1130.052,-90.388,-46.027,178.706,6.157,149.492
C02924=1130.058,-90.639,-46.017,178.704,6.156,149.493
C02925=1130.062,-90.888,-46.008,178.701,6.156,149.493
C02926=1130.068,-91.138,-45.999,178.699,6.155,149.494
C02927=1130.073,-91.388,-45.989,178.698,6.155,149.494
C02928=1130.078,-91.637,-45.980,178.695,6.154,149.495
C02929=1130.084,-91.887,-45.970,178.693,6.154,149.495
C02930=1130.089,-92.137,-45.961,178.692,6.154,149.496
C02931=1130.094,-92.386,-45.952,178.689,6.153,149.496
C02932=1130.100,-92.636,-45.942,178.687,6.152,149.497
C02933=1130.105,-92.886,-45.933,178.686,6.152,149.497
C02934=1130.110,-93.136,-45.924,178.683,6.151,149.498
C02935=1130.116,-93.386,-45.914,178.681,6.151,149.498
C02936=1130.121,-93.636,-45.905,178.679,6.151,149.499
C02937=1130.126,-93.885,-45.896,178.677,6.150,149.499
C02938=1130.132,-94.135,-45.887,178.675,6.150,149.500
C02939=1130.137,-94.385,-45.878,178.673,6.150,149.500
C02940=1130.142,-94.635,-45.868,178.671,6.149,149.501
C02941=1130.148,-94.884,-45.860,178.669,6.148,149.501
C02942=1130.154,-95.134,-45.850,178.667,6.147,149.502
C02943=1130.159,-95.384,-45.841,178.665,6.147,149.502
C02944=1130.164,-95.634,-45.832,178.663,6.147,149.503
C02945=1130.169,-95.883,-45.823,178.661,6.146,149.503
C02946=1130.175,-96.133,-45.813,178.659,6.146,149.504
C02947=1130.180,-96.383,-45.804,178.657,6.145,149.504
C02948=1130.185,-96.633,-45.796,178.655,6.144,149.505
C02949=1130.191,-96.883,-45.786,178.653,6.144,149.505
C02950=1130.196,-97.133,-45.777,178.651,6.144,149.506
C02951=1130.202,-97.383,-45.768,178.649,6.143,149.506
C02952=1130.207,-97.632,-45.759,178.647,6.143,149.507
C02953=1130.213,-97.881,-45.750,178.645,6.142,149.507
C02954=1130.218,-98.131,-45.741,178.643,6.142,149.508
C02955=1130.223,-98.381,-45.732,178.641,6.142,149.508
C02956=1130.229,-98.631,-45.723,178.638,6.141,149.509
C02957=1130.234,-98.881,-45.714,178.636,6.140,149.509
C02958=1130.240,-99.131,-45.704,178.635,6.141,149.510
C02959=1130.245,-99.381,-45.696,178.632,6.140,149.510
C02960=1130.250,-99.631,-45.687,178.630,6.139,149.511
C02961=1130.256,-99.880,-45.678,178.629,6.139,149.511
C02962=1130.261,-100.130,-45.669,178.626,6.138,149.512
C02963=1130.267,-100.380,-45.660,178.625,6.138,149.512
C02964=1130.272,-100.629,-45.650,178.623,6.138,149.513
C02965=1130.277,-100.879,-45.641,178.620,6.137,149.513
C02966=1130.282,-101.129,-45.632,178.619,6.137,149.514
C02967=1130.287,-101.379,-45.623,178.617,6.136,149.514
C02968=1130.294,-101.628,-45.614,178.614,6.135,149.515
C02969=1130.299,-101.878,-45.605,178.613,6.135,149.515
C02970=1130.304,-102.128,-45.597,178.611,6.135,149.516
C02971=1130.309,-102.378,-45.588,178.608,6.134,149.516
C02972=1130.314,-102.627,-45.579,178.607,6.134,149.516
C02973=1130.320,-102.900,-45.569,178.605,6.133,149.517
C02974=1130.326,-103.173,-45.560,178.602,6.133,149.517
C02975=1130.332,-103.444,-45.550,178.600,6.132,149.518
C02976=1130.338,-103.716,-45.540,178.598,6.132,149.519
C02977=1130.343,-103.966,-45.531,178.596,6.131,149.519
C02978=1130.349,-104.216,-45.522,178.594,6.131,149.520
C02979=1130.354,-104.466,-45.513,178.592,6.131,149.520
C02980=1130.359,-104.716,-45.504,178.590,6.130,149.521
C02981=1130.365,-104.965,-45.496,178.588,6.129,149.521
C02982=1130.370,-105.216,-45.487,178.586,6.129,149.522
C02983=1130.376,-105.465,-45.479,178.584,6.129,149.522
C02984=1130.381,-105.715,-45.470,178.582,6.129,149.523
C02985=1130.386,-105.965,-45.461,178.580,6.128,149.523
C02986=1130.392,-106.214,-45.452,178.578,6.127,149.524
C02987=1130.397,-106.464,-45.443,178.576,6.127,149.524
C02988=1130.402,-106.714,-45.434,178.574,6.126,149.525
C02989=1130.407,-106.964,-45.426,178.572,6.126,149.525
C02990=1130.414,-107.213,-45.416,178.570,6.126,149.525
C02991=1130.419,-107.463,-45.407,178.568,6.125,149.526
C02992=1130.424,-107.714,-45.399,178.567,6.125,149.526
C02993=1130.430,-107.964,-45.390,178.564,6.124,149.527
C02994=1130.435,-108.213,-45.382,178.562,6.124,149.527
C02995=1130.440,-108.463,-45.373,178.561,6.124,149.528
C02996=1130.446,-108.712,-45.364,178.558,6.123,149.528
C02997=1130.451,-108.962,-45.355,178.557,6.123,149.529
C02998=1130.456,-109.213,-45.347,178.555,6.122,149.529
C02999=1130.462,-109.462,-45.338,178.552,6.121,149.530
C03000=1130.467,-109.712,-45.330,178.551,6.121,149.530
C03001=1130.472,-109.962,-45.321,178.549,6.121,149.531
C03002=1130.478,-110.211,-45.312,178.547,6.121,149.531
C03003=1130.483,-110.461,-45.303,178.545,6.120,149.532
C03004=1130.489,-110.711,-45.295,178.543,6.119,149.532
C03005=1130.494,-110.961,-45.286,178.542,6.119,149.533
C03006=1130.500,-111.210,-45.278,178.539,6.118,149.533
C03007=1130.505,-111.460,-45.269,178.538,6.118,149.534
C03008=1130.510,-111.710,-45.261,178.536,6.117,149.534
C03009=1130.515,-111.960,-45.252,178.533,6.117,149.535
C03010=1130.521,-112.209,-45.243,178.532,6.117,149.535
C03011=1130.526,-112.459,-45.234,178.530,6.116,149.535
C03012=1130.532,-112.710,-45.226,178.528,6.116,149.536
C03013=1130.538,-112.959,-45.218,178.526,6.115,149.536
C03014=1130.543,-113.209,-45.209,178.524,6.115,149.537
C03015=1130.547,-113.458,-45.200,178.522,6.115,149.537
C03016=1130.553,-113.709,-45.192,178.520,6.114,149.538
C03017=1130.559,-113.958,-45.184,178.518,6.114,149.538
C03018=1130.564,-114.208,-45.175,178.516,6.113,149.539
C03019=1130.569,-114.458,-45.167,178.514,6.113,149.539
C03020=1130.575,-114.707,-45.158,178.512,6.113,149.540
C03021=1130.580,-114.957,-45.149,178.510,6.112,149.540
C03022=1130.586,-115.208,-45.141,178.508,6.112,149.541
C03023=1130.591,-115.457,-45.132,178.506,6.111,149.541
C03024=1130.596,-115.707,-45.123,178.505,6.111,149.542
C03025=1130.602,-115.957,-45.115,178.502,6.110,149.542
C03026=1130.608,-116.206,-45.107,178.501,6.110,149.543
C03027=1130.613,-116.456,-45.098,178.499,6.110,149.543
C03028=1130.618,-116.706,-45.090,178.497,6.109,149.544
C03029=1130.623,-116.955,-45.082,178.495,6.109,149.544
C03030=1130.629,-117.205,-45.073,178.493,6.108,149.545
C03031=1130.635,-117.455,-45.065,178.491,6.108,149.545
C03032=1130.640,-117.705,-45.056,178.489,6.107,149.546
C03033=1130.645,-117.955,-45.048,178.488,6.107,149.546
C03034=1130.651,-118.204,-45.039,178.485,6.106,149.546
C03035=1130.655,-118.454,-45.031,178.483,6.106,149.547
C03036=1130.661,-118.705,-45.023,178.482,6.106,149.547
C03037=1130.667,-118.954,-45.014,178.479,6.105,149.548
C03038=1130.672,-119.204,-45.006,178.478,6.105,149.548
C03039=1130.677,-119.454,-44.997,178.476,6.104,149.549
C03040=1130.683,-119.704,-44.990,178.474,6.104,149.549
C03041=1130.688,-119.953,-44.981,178.472,6.104,149.550
C03042=1130.694,-120.202,-44.973,178.471,6.103,149.550
C03043=1130.699,-120.453,-44.964,178.469,6.103,149.551
C03044=1130.704,-120.703,-44.956,178.467,6.103,149.551
C03045=1130.710,-120.953,-44.948,178.465,6.102,149.552
C03046=1130.715,-121.202,-44.939,178.463,6.101,149.552
C03047=1130.721,-121.452,-44.932,178.461,6.101,149.553
C03048=1130.726,-121.702,-44.923,178.459,6.100,149.553
C03049=1130.731,-121.952,-44.915,178.457,6.101,149.554
C03050=1130.737,-122.201,-44.906,178.455,6.100,149.554
C03051=1130.742,-122.451,-44.898,178.453,6.100,149.555
C03052=1130.748,-122.701,-44.890,178.451,6.099,149.555
C03053=1130.753,-122.951,-44.882,178.450,6.099,149.556
C03054=1130.758,-123.201,-44.873,178.448,6.098,149.556
C03055=1130.764,-123.451,-44.865,178.446,6.098,149.556
C03056=1130.769,-123.700,-44.857,178.444,6.097,149.557
C03057=1130.775,-123.950,-44.849,178.443,6.097,149.557
C03058=1130.780,-124.200,-44.840,178.440,6.097,149.558
C03059=1130.786,-124.450,-44.832,178.438,6.096,149.558
C03060=1130.791,-124.700,-44.825,178.437,6.096,149.559
C03061=1130.796,-124.950,-44.816,178.434,6.095,149.559
C03062=1130.802,-125.199,-44.808,178.433,6.095,149.560
C03063=1130.807,-125.449,-44.800,178.431,6.094,149.560
C03064=1130.813,-125.699,-44.792,178.429,6.094,149.560
C03065=1130.818,-125.949,-44.783,178.427,6.093,149.561
C03066=1130.824,-126.198,-44.775,178.426,6.093,149.561
C03067=1130.829,-126.449,-44.767,178.423,6.093,149.562
C03068=1130.834,-126.698,-44.759,178.422,6.093,149.562
C03069=1130.840,-126.948,-44.751,178.420,6.092,149.563
C03070=1130.845,-127.197,-44.743,178.418,6.092,149.563
C03071=1130.850,-127.447,-44.735,178.416,6.091,149.564
C03072=1130.856,-127.697,-44.727,178.415,6.091,149.564
C03073=1130.861,-127.947,-44.719,178.413,6.090,149.565
C03074=1130.867,-128.196,-44.711,178.411,6.090,149.565
C03075=1130.872,-128.447,-44.703,178.409,6.090,149.566
C03076=1130.878,-128.696,-44.694,178.407,6.090,149.566
C03077=1130.457,-128.708,-44.739,178.404,6.093,149.568
C03078=1130.451,-128.458,-44.747,178.405,6.094,149.567
C03079=1130.446,-128.208,-44.755,178.407,6.094,149.567
C03080=1130.441,-127.959,-44.763,178.409,6.094,149.566
C03081=1130.435,-127.708,-44.771,178.411,6.094,149.566
C03082=1130.429,-127.459,-44.779,178.413,6.095,149.565
C03083=1130.425,-127.209,-44.787,178.415,6.095,149.565
C03084=1130.419,-126.959,-44.795,178.417,6.096,149.564
C03085=1130.414,-126.709,-44.804,178.418,6.096,149.564
C03086=1130.408,-126.460,-44.812,178.420,6.097,149.564
C03087=1130.403,-126.209,-44.819,178.422,6.097,149.563
C03088=1130.397,-125.960,-44.828,178.424,6.098,149.563
C03089=1130.392,-125.710,-44.836,178.426,6.097,149.562
C03090=1130.387,-125.461,-44.844,178.428,6.098,149.562
C03091=1130.381,-125.211,-44.852,178.429,6.098,149.561
C03092=1130.376,-124.960,-44.860,178.432,6.099,149.561
C03093=1130.370,-124.711,-44.869,178.434,6.100,149.560
C03094=1130.365,-124.461,-44.876,178.435,6.100,149.560
C03095=1130.359,-124.212,-44.885,178.437,6.101,149.560
C03096=1130.354,-123.961,-44.893,178.439,6.101,149.559
C03097=1130.348,-123.712,-44.902,178.441,6.101,149.559
C03098=1130.343,-123.462,-44.909,178.442,6.101,149.558
C03099=1130.338,-123.212,-44.918,178.445,6.102,149.558
C03100=1130.332,-122.962,-44.926,178.446,6.102,149.557
C03101=1130.327,-122.712,-44.934,178.448,6.103,149.557
C03102=1130.322,-122.463,-44.942,178.450,6.103,149.556
C03103=1130.316,-122.212,-44.950,178.452,6.104,149.556
C03104=1130.310,-121.963,-44.959,178.453,6.104,149.555
C03105=1130.305,-121.713,-44.967,178.456,6.105,149.555
C03106=1130.300,-121.463,-44.976,178.457,6.105,149.554
C03107=1130.294,-121.213,-44.983,178.459,6.105,149.554
C03108=1130.289,-120.964,-44.992,178.462,6.106,149.553
C03109=1130.283,-120.714,-45.000,178.463,6.106,149.553
C03110=1130.278,-120.464,-45.009,178.465,6.107,149.552
C03111=1130.273,-120.214,-45.018,178.467,6.107,149.552
C03112=1130.268,-119.965,-45.025,178.469,6.107,149.551
C03113=1130.262,-119.715,-45.034,178.471,6.107,149.551
C03114=1130.256,-119.465,-45.041,178.473,6.108,149.550
C03115=1130.251,-119.215,-45.050,178.474,6.108,149.550
C03116=1130.246,-118.965,-45.059,178.476,6.109,149.550
C03117=1130.241,-118.716,-45.066,178.478,6.110,149.549
C03118=1130.235,-118.466,-45.075,178.480,6.110,149.549
C03119=1130.230,-118.216,-45.084,178.482,6.111,149.548
C03120=1130.224,-117.966,-45.092,178.484,6.111,149.548
C03121=1130.219,-117.716,-45.100,178.486,6.111,149.547
C03122=1130.214,-117.466,-45.109,178.488,6.111,149.547
C03123=1130.208,-117.217,-45.118,178.490,6.112,149.546
C03124=1130.202,-116.967,-45.126,178.491,6.112,149.546
C03125=1130.197,-116.718,-45.134,178.494,6.113,149.545
C03126=1130.192,-116.467,-45.142,178.496,6.113,149.545
C03127=1130.187,-116.217,-45.151,178.497,6.113,149.544
C03128=1130.181,-115.968,-45.159,178.500,6.114,149.544
C03129=1130.175,-115.718,-45.168,178.501,6.114,149.544
C03130=1130.170,-115.468,-45.177,178.503,6.115,149.543
C03131=1130.164,-115.219,-45.185,178.505,6.115,149.543
C03132=1130.159,-114.968,-45.193,178.507,6.116,149.542
C03133=1130.154,-114.718,-45.202,178.509,6.117,149.542
C03134=1130.148,-114.469,-45.211,178.511,6.117,149.541
C03135=1130.143,-114.219,-45.218,178.513,6.117,149.541
C03136=1130.138,-113.969,-45.227,178.514,6.117,149.540
C03137=1130.132,-113.720,-45.236,178.517,6.118,149.540
C03138=1130.127,-113.470,-45.245,178.519,6.119,149.539
C03139=1130.122,-113.220,-45.253,178.520,6.119,149.539
C03140=1130.117,-112.970,-45.262,178.523,6.119,149.538
C03141=1130.111,-112.721,-45.270,178.524,6.119,149.538
C03142=1130.105,-112.470,-45.278,178.526,6.120,149.537
C03143=1130.100,-112.220,-45.287,178.528,6.120,149.537
C03144=1130.094,-111.971,-45.296,178.530,6.121,149.536
C03145=1130.089,-111.721,-45.305,178.532,6.122,149.536
C03146=1130.084,-111.471,-45.313,178.534,6.122,149.535
C03147=1130.079,-111.221,-45.322,178.536,6.122,149.535
C03148=1130.073,-110.972,-45.330,178.538,6.122,149.534
C03149=1130.068,-110.722,-45.339,178.540,6.123,149.534
C03150=1130.063,-110.472,-45.348,178.542,6.124,149.533
C03151=1130.056,-110.223,-45.356,178.544,6.124,149.533
C03152=1130.051,-109.973,-45.365,178.545,6.125,149.533
C03153=1130.046,-109.723,-45.374,178.547,6.125,149.532
C03154=1130.041,-109.473,-45.383,178.549,6.125,149.532
C03155=1130.035,-109.224,-45.391,178.551,6.126,149.531
C03156=1130.030,-108.973,-45.399,178.553,6.126,149.531
C03157=1130.025,-108.723,-45.408,178.555,6.127,149.530
C03158=1130.019,-108.474,-45.417,178.557,6.127,149.530
C03159=1130.014,-108.224,-45.426,178.559,6.128,149.529
C03160=1130.008,-107.975,-45.435,178.561,6.128,149.529
C03161=1130.003,-107.725,-45.443,178.563,6.128,149.528
C03162=1129.998,-107.474,-45.452,178.565,6.129,149.528
C03163=1129.992,-107.225,-45.460,178.567,6.129,149.527
C03164=1129.987,-106.975,-45.469,178.569,6.130,149.527
C03165=1129.982,-106.725,-45.478,178.571,6.131,149.526
C03166=1129.977,-106.476,-45.487,178.573,6.130,149.526
C03167=1129.971,-106.226,-45.496,178.575,6.131,149.525
C03168=1129.966,-105.977,-45.504,178.577,6.132,149.525
C03169=1129.960,-105.726,-45.514,178.579,6.132,149.524
C03170=1129.955,-105.477,-45.523,178.581,6.133,149.524
C03171=1129.949,-105.226,-45.531,178.582,6.133,149.523
C03172=1129.944,-104.976,-45.540,178.585,6.133,149.523
C03173=1129.938,-104.727,-45.548,178.587,6.134,149.522
C03174=1129.933,-104.477,-45.557,178.588,6.134,149.522
C03175=1129.928,-104.227,-45.566,178.591,6.135,149.521
C03176=1129.923,-103.978,-45.575,178.593,6.136,149.521
C03177=1129.917,-103.728,-45.584,178.594,6.135,149.520
C03178=1129.912,-103.455,-45.593,178.597,6.136,149.520
C03179=1129.906,-103.184,-45.603,178.599,6.137,149.519
C03180=1129.900,-102.911,-45.613,178.601,6.137,149.519
C03181=1129.893,-102.639,-45.623,178.603,6.137,149.518
C03182=1129.888,-102.389,-45.632,178.605,6.138,149.518
C03183=1129.883,-102.139,-45.641,178.607,6.139,149.517
C03184=1129.878,-101.889,-45.650,178.609,6.139,149.517
C03185=1129.873,-101.639,-45.658,178.611,6.139,149.516
C03186=1129.867,-101.390,-45.667,178.613,6.140,149.516
C03187=1129.862,-101.140,-45.676,178.615,6.140,149.515
C03188=1129.856,-100.890,-45.685,178.617,6.141,149.515
C03189=1129.851,-100.640,-45.694,178.619,6.142,149.514
C03190=1129.845,-100.390,-45.703,178.621,6.142,149.514
C03191=1129.840,-100.140,-45.712,178.623,6.142,149.513
C03192=1129.834,-99.891,-45.721,178.625,6.142,149.513
C03193=1129.829,-99.642,-45.731,178.627,6.143,149.512
C03194=1129.824,-99.392,-45.740,178.629,6.144,149.512
C03195=1129.819,-99.142,-45.749,178.631,6.144,149.512
C03196=1129.813,-98.892,-45.758,178.633,6.145,149.511
C03197=1129.808,-98.642,-45.766,178.635,6.145,149.511
C03198=1129.802,-98.392,-45.776,178.637,6.145,149.510
C03199=1129.797,-98.142,-45.785,178.639,6.146,149.510
C03200=1129.791,-97.893,-45.793,178.641,6.147,149.509
C03201=1129.786,-97.643,-45.802,178.643,6.147,149.509
C03202=1129.780,-97.393,-45.812,178.645,6.147,149.508
C03203=1129.775,-97.144,-45.821,178.648,6.148,149.507
C03204=1129.770,-96.894,-45.830,178.649,6.148,149.507
C03205=1129.765,-96.644,-45.839,178.651,6.148,149.506
C03206=1129.759,-96.394,-45.849,178.654,6.149,149.506
C03207=1129.754,-96.144,-45.858,178.655,6.149,149.505
C03208=1129.749,-95.894,-45.866,178.657,6.150,149.505
C03209=1129.744,-95.644,-45.875,178.660,6.151,149.504
C03210=1129.738,-95.395,-45.886,178.661,6.151,149.504
C03211=1129.732,-95.146,-45.894,178.663,6.151,149.504
C03212=1129.727,-94.896,-45.903,178.666,6.152,149.503
C03213=1129.721,-94.646,-45.912,178.667,6.152,149.503
C03214=1129.716,-94.396,-45.921,178.669,6.153,149.502
C03215=1129.711,-94.147,-45.931,178.672,6.154,149.502
C03216=1129.706,-93.897,-45.940,178.674,6.154,149.501
C03217=1129.700,-93.647,-45.949,178.675,6.154,149.501
C03218=1129.695,-93.397,-45.958,178.678,6.155,149.500
C03219=1129.690,-93.148,-45.968,178.680,6.156,149.500
C03220=1129.684,-92.897,-45.977,178.681,6.156,149.499
C03221=1129.679,-92.648,-45.986,178.684,6.157,149.499
C03222=1129.674,-92.398,-45.995,178.686,6.157,149.498
C03223=1129.668,-92.148,-46.005,178.688,6.157,149.497
C03224=1129.663,-91.898,-46.014,178.690,6.158,149.497
C03225=1129.658,-91.648,-46.023,178.692,6.158,149.496
C03226=1129.652,-91.398,-46.033,178.694,6.158,149.496
C03227=1129.647,-91.149,-46.042,178.696,6.159,149.496
C03228=1129.642,-90.899,-46.051,178.698,6.160,149.495
C03229=1129.636,-90.649,-46.061,178.700,6.161,149.495
C03230=1129.631,-90.400,-46.070,178.702,6.160,149.494
C03231=1129.625,-90.150,-46.080,178.704,6.161,149.494
C03232=1129.620,-89.900,-46.089,178.706,6.162,149.493
C03233=1129.615,-89.651,-46.098,178.708,6.162,149.493
C03234=1129.609,-89.400,-46.108,178.710,6.163,149.492
C03235=1129.604,-89.151,-46.117,178.712,6.163,149.492
C03236=1129.599,-88.901,-46.127,178.715,6.164,149.491
C03237=1129.593,-88.651,-46.136,178.717,6.164,149.490
C03238=1129.588,-88.401,-46.145,178.719,6.165,149.490
C03239=1129.583,-88.152,-46.155,178.721,6.165,149.489
C03240=1129.578,-87.902,-46.164,178.723,6.165,149.489
C03241=1129.572,-87.652,-46.173,178.725,6.166,149.489
C03242=1129.567,-87.403,-46.183,178.727,6.167,149.488
C03243=1129.562,-87.153,-46.192,178.729,6.167,149.488
C03244=1129.556,-86.903,-46.202,178.731,6.167,149.487
C03245=1129.551,-86.653,-46.211,178.733,6.168,149.487
C03246=1129.545,-86.403,-46.220,178.735,6.169,149.486
C03247=1129.540,-86.154,-46.230,178.737,6.169,149.486
C03248=1129.534,-85.904,-46.239,178.739,6.170,149.485
C03249=1129.529,-85.655,-46.249,178.742,6.170,149.484
C03250=1129.523,-85.404,-46.259,178.744,6.171,149.484
C03251=1129.519,-85.155,-46.268,178.745,6.171,149.483
C03252=1129.513,-84.905,-46.277,178.748,6.171,149.483
C03253=1129.508,-84.656,-46.287,178.750,6.172,149.482
C03254=1129.503,-84.405,-46.297,178.752,6.173,149.482
C03255=1129.498,-84.156,-46.307,178.754,6.173,149.481
C03256=1129.492,-83.906,-46.316,178.756,6.174,149.481
C03257=1129.487,-83.656,-46.326,178.758,6.174,149.481
C03258=1129.482,-83.406,-46.335,178.760,6.175,149.480
C03259=1129.476,-83.157,-46.345,178.762,6.175,149.480
C03260=1129.471,-82.907,-46.354,178.764,6.176,149.479
C03261=1129.465,-82.657,-46.364,178.767,6.176,149.478
C03262=1129.459,-82.407,-46.374,178.769,6.177,149.478
C03263=1129.455,-82.158,-46.383,178.770,6.177,149.477
C03264=1129.449,-81.908,-46.393,178.773,6.178,149.477
C03265=1129.444,-81.658,-46.403,178.775,6.179,149.476
C03266=1129.439,-81.408,-46.412,178.777,6.179,149.476
C03267=1129.434,-81.159,-46.422,178.779,6.179,149.475
C03268=1129.428,-80.908,-46.431,178.781,6.180,149.475
C03269=1129.423,-80.659,-46.441,178.784,6.180,149.474
C03270=1129.417,-80.410,-46.451,178.786,6.181,149.474
C03271=1129.411,-80.159,-46.461,178.787,6.181,149.473
C03272=1129.407,-79.910,-46.470,178.790,6.182,149.473
C03273=1129.401,-79.659,-46.480,178.792,6.183,149.472
C03274=1129.396,-79.410,-46.490,178.794,6.183,149.472
C03275=1129.391,-79.161,-46.500,178.795,6.183,149.471
C03276=1129.385,-78.910,-46.509,178.798,6.184,149.471
C03277=1129.380,-78.661,-46.519,178.800,6.185,149.470
C03278=1129.374,-78.411,-46.528,178.803,6.185,149.470
C03279=1129.369,-78.162,-46.538,178.804,6.185,149.469
C03280=1129.364,-77.912,-46.548,178.806,6.186,149.469
C03281=1129.358,-77.661,-46.558,178.809,6.187,149.468
C03282=1129.353,-77.391,-46.569,178.811,6.187,149.468
C03283=1129.347,-77.119,-46.579,178.813,6.188,149.467
C03284=1129.341,-76.847,-46.591,178.816,6.188,149.467
C03285=1129.336,-76.575,-46.601,178.818,6.189,149.466
C03286=1129.330,-76.326,-46.611,178.820,6.190,149.466
C03287=1129.324,-76.076,-46.621,178.822,6.190,149.465
C03288=1129.319,-75.826,-46.630,178.824,6.190,149.464
C03289=1129.314,-75.577,-46.640,178.826,6.191,149.464
C03290=1129.308,-75.327,-46.650,178.829,6.192,149.463
C03291=1129.304,-75.077,-46.660,178.830,6.192,149.463
C03292=1129.298,-74.827,-46.670,178.832,6.193,149.462
C03293=1129.292,-74.578,-46.680,178.835,6.193,149.462
C03294=1129.287,-74.328,-46.690,178.837,6.194,149.461
C03295=1129.282,-74.079,-46.700,178.839,6.195,149.461
C03296=1129.277,-73.828,-46.710,178.841,6.194,149.460
C03297=1129.271,-73.579,-46.720,178.843,6.195,149.460
C03298=1129.266,-73.329,-46.730,178.845,6.196,149.459
C03299=1129.260,-73.080,-46.740,178.848,6.197,149.459
C03300=1129.255,-72.830,-46.749,178.850,6.197,149.458
C03301=1129.250,-72.580,-46.759,178.851,6.197,149.458
C03302=1129.245,-72.330,-46.770,178.854,6.198,149.457
C03303=1129.239,-72.081,-46.780,178.856,6.199,149.457
C03304=1129.234,-71.831,-46.790,178.859,6.199,149.456
C03305=1129.229,-71.581,-46.800,178.861,6.200,149.456
C03306=1129.223,-71.331,-46.809,178.862,6.200,149.455
C03307=1129.218,-71.081,-46.820,178.864,6.201,149.455
C03308=1129.212,-70.832,-46.830,178.867,6.202,149.454
C03309=1129.207,-70.582,-46.840,178.869,6.202,149.454
C03310=1129.202,-70.332,-46.850,178.872,6.203,149.453
C03311=1129.197,-70.083,-46.860,178.874,6.203,149.453
C03312=1129.191,-69.833,-46.870,178.875,6.203,149.452
C03313=1129.186,-69.582,-46.880,178.878,6.204,149.452
C03314=1129.181,-69.333,-46.890,178.880,6.205,149.451
C03315=1129.175,-69.084,-46.900,178.882,6.206,149.451
C03316=1129.170,-68.833,-46.911,178.885,6.206,149.450
C03317=1129.165,-68.584,-46.921,178.886,6.206,149.450
C03318=1129.159,-68.334,-46.931,178.888,6.207,149.449
C03319=1129.154,-68.085,-46.941,178.891,6.208,149.449
C03320=1129.149,-67.835,-46.951,178.893,6.208,149.448
C03321=1129.144,-67.585,-46.962,178.895,6.209,149.448
C03322=1129.138,-67.336,-46.972,178.898,6.209,149.447
C03323=1129.133,-67.085,-46.982,178.899,6.209,149.446
C03324=1129.128,-66.836,-46.993,178.901,6.210,149.446
C03325=1129.122,-66.586,-47.003,178.904,6.211,149.445
C03326=1129.118,-66.336,-47.013,178.906,6.212,149.445
C03327=1129.112,-66.087,-47.023,178.908,6.212,149.444
C03328=1129.106,-65.837,-47.033,178.910,6.213,149.444
C03329=1129.101,-65.587,-47.044,178.913,6.214,149.443
C03330=1129.096,-65.338,-47.054,178.914,6.214,149.443
C03331=1129.090,-65.088,-47.064,178.917,6.214,149.442
C03332=1129.085,-64.838,-47.075,178.919,6.215,149.442
C03333=1129.080,-64.588,-47.085,178.921,6.216,149.441
C03334=1129.074,-64.339,-47.095,178.923,6.217,149.441
C03335=1129.070,-64.089,-47.105,178.926,6.217,149.440
C03336=1129.064,-63.839,-47.115,178.927,6.217,149.440
C03337=1129.059,-63.590,-47.125,178.930,6.218,149.439
C03338=1129.054,-63.339,-47.136,178.932,6.218,149.439
C03339=1129.048,-63.090,-47.146,178.934,6.219,149.438
C03340=1129.042,-62.840,-47.156,178.937,6.220,149.438
C03341=1129.037,-62.590,-47.167,178.939,6.220,149.437
C03342=1129.032,-62.341,-47.177,178.941,6.221,149.437
C03343=1129.027,-62.091,-47.189,178.943,6.221,149.436
C03344=1129.022,-61.841,-47.199,178.945,6.222,149.436
C03345=1129.016,-61.592,-47.209,178.947,6.223,149.435
C03346=1129.011,-61.342,-47.220,178.950,6.223,149.434
C03347=1129.005,-61.092,-47.230,178.952,6.224,149.434
C03348=1129.000,-60.842,-47.240,178.954,6.224,149.433
C03349=1128.995,-60.592,-47.251,178.956,6.225,149.433
C03350=1128.989,-60.343,-47.261,178.959,6.226,149.432
C03351=1128.984,-60.093,-47.272,178.961,6.226,149.432
C03352=1128.979,-59.844,-47.282,178.963,6.226,149.431
C03353=1128.974,-59.593,-47.293,178.965,6.227,149.431
C03354=1128.968,-59.344,-47.303,178.967,6.228,149.430
C03355=1128.963,-59.094,-47.314,178.969,6.229,149.430
C03356=1128.958,-58.845,-47.325,178.972,6.229,149.429
C03357=1128.952,-58.595,-47.335,178.974,6.230,149.429
C03358=1128.947,-58.345,-47.345,178.976,6.231,149.428
C03359=1128.942,-58.095,-47.356,178.979,6.231,149.428
C03360=1128.937,-57.846,-47.367,178.980,6.231,149.427
C03361=1128.931,-57.596,-47.377,178.982,6.232,149.427
C03362=1128.926,-57.346,-47.388,178.985,6.232,149.426
C03363=1128.921,-57.096,-47.398,178.987,6.233,149.426
C03364=1128.916,-56.847,-47.409,178.989,6.234,149.425
C03365=1128.911,-56.597,-47.419,178.992,6.235,149.425
C03366=1128.906,-56.347,-47.430,178.994,6.235,149.424
C03367=1128.900,-56.097,-47.440,178.997,6.236,149.423
C03368=1128.895,-55.848,-47.451,178.999,6.237,149.423
C03369=1128.890,-55.598,-47.462,179.001,6.237,149.422
C03370=1128.884,-55.349,-47.472,179.002,6.237,149.422
C03371=1128.879,-55.099,-47.483,179.005,6.238,149.421
C03372=1128.874,-54.850,-47.493,179.007,6.238,149.421
C03373=1128.869,-54.599,-47.504,179.010,6.239,149.420
C03374=1128.863,-54.350,-47.515,179.012,6.240,149.420
C03375=1128.858,-54.100,-47.526,179.014,6.241,149.419
C03376=1128.852,-53.850,-47.536,179.016,6.242,149.419
C03377=1128.848,-53.601,-47.547,179.019,6.242,149.418
C03378=1128.842,-53.351,-47.558,179.021,6.243,149.418
C03379=1128.837,-53.101,-47.568,179.023,6.243,149.417
C03380=1128.832,-52.852,-47.579,179.025,6.244,149.417
C03381=1128.827,-52.602,-47.590,179.028,6.245,149.416
C03382=1128.821,-52.352,-47.602,179.030,6.245,149.416
C03383=1128.816,-52.102,-47.612,179.032,6.245,149.415
C03384=1128.811,-51.852,-47.622,179.034,6.246,149.415
C03385=1128.805,-51.603,-47.633,179.036,6.247,149.414
C03386=1128.800,-51.332,-47.646,179.039,6.247,149.413
C03387=1128.793,-51.061,-47.657,179.041,6.248,149.413
C03388=1128.788,-50.790,-47.668,179.044,6.250,149.412
C03389=1128.783,-50.519,-47.681,179.047,6.250,149.412
C03390=1128.777,-50.270,-47.691,179.049,6.251,149.411
C03391=1128.772,-50.020,-47.702,179.050,6.251,149.411
C03392=1128.766,-49.770,-47.713,179.052,6.251,149.410
C03393=1128.761,-49.521,-47.724,179.055,6.252,149.410
C03394=1128.756,-49.271,-47.734,179.057,6.253,149.409
C03395=1128.751,-49.022,-47.746,179.060,6.253,149.409
C03396=1128.745,-48.771,-47.757,179.062,6.254,149.408
C03397=1128.740,-48.522,-47.768,179.064,6.255,149.407
C03398=1128.735,-48.272,-47.778,179.067,6.255,149.407
C03399=1128.730,-48.023,-47.789,179.069,6.256,149.406
C03400=1128.724,-47.772,-47.801,179.071,6.257,149.406
C03401=1128.719,-47.523,-47.812,179.073,6.258,149.406
C03402=1128.714,-47.273,-47.822,179.076,6.258,149.405
C03403=1128.709,-47.024,-47.833,179.078,6.259,149.404
C03404=1128.703,-46.774,-47.844,179.080,6.260,149.404
C03405=1128.698,-46.524,-47.855,179.082,6.260,149.403
C03406=1128.693,-46.275,-47.867,179.085,6.261,149.403
C03407=1128.687,-46.025,-47.877,179.087,6.261,149.402
C03408=1128.682,-45.775,-47.889,179.089,6.262,149.402
C03409=1128.677,-45.526,-47.899,179.092,6.263,149.401
C03410=1128.671,-45.276,-47.911,179.094,6.264,149.401
C03411=1128.667,-45.026,-47.922,179.096,6.264,149.400
C03412=1128.661,-44.776,-47.932,179.099,6.265,149.400
C03413=1128.656,-44.527,-47.944,179.101,6.266,149.399
C03414=1128.651,-44.277,-47.956,179.103,6.266,149.399
C03415=1128.645,-44.027,-47.966,179.105,6.266,149.398
C03416=1128.640,-43.777,-47.978,179.107,6.267,149.397
C03417=1128.635,-43.528,-47.989,179.109,6.268,149.397
C03418=1128.630,-43.278,-47.999,179.112,6.268,149.397
C03419=1128.624,-43.028,-48.011,179.114,6.269,149.396
C03420=1128.619,-42.779,-48.022,179.117,6.270,149.395
C03421=1128.614,-42.529,-48.033,179.119,6.270,149.395
C03422=1128.608,-42.279,-48.044,179.121,6.271,149.394
C03423=1128.604,-42.030,-48.056,179.123,6.272,149.394
C03424=1128.598,-41.780,-48.066,179.126,6.272,149.393
C03425=1128.593,-41.530,-48.078,179.128,6.273,149.393
C03426=1128.588,-41.280,-48.089,179.130,6.274,149.392
C03427=1128.582,-41.031,-48.101,179.132,6.275,149.392
C03428=1128.577,-40.781,-48.111,179.135,6.275,149.391
C03429=1128.572,-40.531,-48.122,179.137,6.276,149.391
C03430=1128.566,-40.282,-48.134,179.139,6.276,149.390
C03431=1128.562,-40.032,-48.145,179.142,6.277,149.390
C03432=1128.556,-39.783,-48.157,179.144,6.278,149.389
C03433=1128.550,-39.533,-48.167,179.146,6.278,149.388
C03434=1128.545,-39.283,-48.179,179.149,6.279,149.388
C03435=1128.540,-39.033,-48.191,179.151,6.280,149.388
C03436=1128.535,-38.783,-48.202,179.153,6.281,149.387
C03437=1128.530,-38.535,-48.213,179.156,6.281,149.386
C03438=1128.524,-38.284,-48.225,179.158,6.282,149.386
C03439=1128.519,-38.034,-48.236,179.160,6.283,149.385
C03440=1128.514,-37.784,-48.248,179.162,6.283,149.385
C03441=1128.508,-37.536,-48.259,179.165,6.284,149.384
C03442=1128.483,-36.347,-48.313,179.529,5.660,149.141
C03443=1128.478,-36.097,-48.325,179.530,5.665,149.142
C03444=1128.473,-35.847,-48.336,179.531,5.669,149.142
C03445=1128.468,-35.597,-48.348,179.532,5.674,149.143
C03446=1128.463,-35.348,-48.359,179.533,5.679,149.144
C03447=1128.457,-35.098,-48.371,179.534,5.684,149.145
C03448=1128.453,-34.849,-48.382,179.534,5.688,149.146
C03449=1128.447,-34.598,-48.393,179.534,5.693,149.146
C03450=1128.441,-34.349,-48.404,179.535,5.698,149.147
C03451=1128.434,-33.988,-48.421,179.535,5.704,149.149
C03452=1128.426,-33.626,-48.438,179.537,5.711,149.150
C03453=1128.419,-33.265,-48.455,179.537,5.717,149.151
C03454=1128.412,-32.903,-48.472,179.537,5.723,149.152
C03455=1128.406,-32.653,-48.484,179.537,5.728,149.153
C03456=1128.401,-32.404,-48.495,179.537,5.732,149.154
C03457=1128.395,-32.155,-48.506,179.538,5.737,149.155
C03458=1128.391,-31.905,-48.518,179.537,5.741,149.156
C03459=1128.385,-31.655,-48.530,179.538,5.745,149.157
C03460=1128.380,-31.405,-48.541,179.538,5.749,149.158
C03461=1128.375,-31.155,-48.553,179.538,5.753,149.159
C03462=1128.369,-30.906,-48.564,179.537,5.758,149.160
C03463=1128.364,-30.657,-48.576,179.537,5.762,149.161
C03464=1128.359,-30.407,-48.587,179.537,5.766,149.162
C03465=1128.354,-30.157,-48.599,179.536,5.770,149.163
C03466=1128.349,-29.907,-48.611,179.536,5.774,149.164
C03467=1128.343,-29.657,-48.623,179.535,5.778,149.165
C03468=1128.337,-29.408,-48.634,179.535,5.782,149.166
C03469=1128.333,-29.158,-48.645,179.534,5.786,149.167
C03470=1128.327,-28.908,-48.657,179.534,5.790,149.168
C03471=1128.322,-28.659,-48.670,179.534,5.795,149.169
C03472=1128.317,-28.409,-48.681,179.533,5.798,149.170
C03473=1128.312,-28.159,-48.693,179.532,5.803,149.171
C03474=1128.307,-27.909,-48.705,179.531,5.806,149.172
C03475=1128.302,-27.660,-48.716,179.531,5.810,149.173
C03476=1128.296,-27.411,-48.728,179.529,5.814,149.174
C03477=1128.290,-27.161,-48.740,179.529,5.818,149.175
C03478=1128.286,-26.911,-48.751,179.527,5.821,149.177
C03479=1128.281,-26.662,-48.763,179.526,5.825,149.178
C03480=1128.275,-26.412,-48.775,179.525,5.830,149.179
C03481=1128.271,-26.162,-48.787,179.524,5.833,149.180
C03482=1128.265,-25.912,-48.799,179.523,5.838,149.181
C03483=1128.260,-25.662,-48.810,179.525,5.843,149.182
C03484=1128.255,-25.413,-48.822,179.525,5.848,149.183
C03485=1128.249,-25.163,-48.833,179.526,5.853,149.184
C03486=1128.244,-24.914,-48.846,179.527,5.858,149.185
C03487=1128.239,-24.665,-48.857,179.528,5.863,149.186
C03488=1128.234,-24.415,-48.869,179.529,5.868,149.186
C03489=1128.228,-24.165,-48.881,179.529,5.872,149.187
C03490=1128.223,-23.915,-48.893,179.530,5.878,149.188
C03491=1128.218,-23.665,-48.905,179.531,5.883,149.189
C03492=1128.213,-23.416,-48.917,179.532,5.887,149.190
C03493=1128.208,-23.166,-48.929,179.533,5.893,149.190
C03494=1128.202,-22.917,-48.941,179.533,5.897,149.191
C03495=1128.197,-22.667,-48.953,179.534,5.902,149.192
C03496=1128.192,-22.417,-48.964,179.536,5.907,149.193
C03497=1128.187,-22.167,-48.976,179.536,5.912,149.194
C03498=1128.181,-21.918,-48.988,179.536,5.917,149.195
C03499=1128.176,-21.668,-49.000,179.538,5.922,149.196
C03500=1128.170,-21.419,-49.012,179.539,5.927,149.196
C03501=1128.165,-21.169,-49.025,179.539,5.931,149.197
C03502=1128.160,-20.920,-49.036,179.540,5.937,149.198
C03503=1128.156,-20.704,-49.047,179.540,5.940,149.199
C03504=1128.151,-20.489,-49.058,179.541,5.945,149.199
C03505=1128.147,-20.273,-49.068,179.542,5.949,149.200
C03506=1128.142,-20.057,-49.078,179.542,5.953,149.201
C03507=1128.138,-19.842,-49.088,179.543,5.957,149.202
C03508=1128.134,-19.626,-49.099,179.544,5.962,149.202
C03509=1128.129,-19.410,-49.110,179.545,5.965,149.203
C03510=1128.125,-19.195,-49.120,179.546,5.970,149.203
C03511=1128.119,-18.945,-49.132,179.546,5.974,149.204
C03512=1128.114,-18.696,-49.145,179.547,5.980,149.205
C03513=1128.109,-18.446,-49.157,179.548,5.984,149.206
C03514=1128.104,-18.196,-49.169,179.549,5.989,149.207
C03515=1128.098,-17.946,-49.181,179.549,5.994,149.208
C03516=1128.093,-17.697,-49.194,179.550,5.998,149.209
C03517=1128.088,-17.447,-49.206,179.551,6.004,149.209
C03518=1128.083,-17.198,-49.218,179.552,6.008,149.210
C03519=1128.077,-16.948,-49.230,179.552,6.013,149.211
C03520=1128.072,-16.699,-49.243,179.553,6.017,149.212
C03521=1128.067,-16.449,-49.255,179.554,6.022,149.213
C03522=1128.062,-16.200,-49.267,179.554,6.027,149.213
C03523=1128.057,-15.950,-49.278,179.556,6.032,149.214
C03524=1128.052,-15.700,-49.291,179.556,6.037,149.215
C03525=1128.047,-15.451,-49.304,179.557,6.042,149.216
C03526=1128.042,-15.200,-49.316,179.558,6.046,149.217
C03527=1128.037,-14.951,-49.328,179.558,6.051,149.217
C03528=1128.030,-14.701,-49.341,179.559,6.055,149.218
C03529=1128.025,-14.452,-49.354,179.560,6.060,149.219
C03530=1128.020,-14.202,-49.366,179.561,6.065,149.220
C03531=1128.015,-13.952,-49.378,179.562,6.070,149.221
C03532=1128.010,-13.703,-49.391,179.562,6.074,149.221
C03533=1128.004,-13.454,-49.403,179.563,6.079,149.222
C03534=1128.000,-13.203,-49.415,179.564,6.083,149.223
C03535=1127.995,-12.954,-49.428,179.564,6.088,149.224
C03536=1127.989,-12.704,-49.441,179.565,6.093,149.225
C03537=1127.984,-12.454,-49.453,179.566,6.097,149.225
C03538=1127.979,-12.205,-49.465,179.566,6.102,149.226
C03539=1127.974,-11.956,-49.478,179.567,6.107,149.227
C03540=1127.969,-11.706,-49.491,179.568,6.111,149.228
C03541=1127.964,-11.456,-49.503,179.568,6.116,149.229
C03542=1127.958,-11.206,-49.516,179.569,6.120,149.230
C03543=1127.953,-10.957,-49.528,179.570,6.125,149.230
C03544=1127.948,-10.708,-49.541,179.571,6.130,149.231
C03545=1127.942,-10.458,-49.553,179.572,6.135,149.232
C03546=1127.938,-10.208,-49.566,179.572,6.139,149.233
C03547=1127.933,-9.958,-49.578,179.573,6.144,149.234
C03548=1127.927,-9.709,-49.591,179.574,6.148,149.234
C03549=1127.922,-9.459,-49.604,179.574,6.153,149.235
C03550=1127.917,-9.209,-49.617,179.575,6.158,149.236
C03551=1127.912,-8.959,-49.629,179.576,6.162,149.237
C03552=1127.907,-8.710,-49.642,179.576,6.167,149.238
C03553=1127.901,-8.461,-49.654,179.577,6.172,149.238
C03554=1127.896,-8.212,-49.667,179.578,6.176,149.239
C03555=1127.891,-7.961,-49.680,179.578,6.180,149.240
C03556=1127.886,-7.712,-49.693,179.578,6.185,149.241
C03557=1127.881,-7.463,-49.706,179.579,6.189,149.242
C03558=1127.876,-7.213,-49.718,179.580,6.194,149.242
C03559=1127.871,-6.997,-49.729,179.581,6.198,149.243
C03560=1127.867,-6.781,-49.740,179.581,6.202,149.244
C03561=1127.863,-6.566,-49.752,179.582,6.206,149.244
C03562=1127.857,-6.351,-49.763,179.582,6.210,149.245
C03563=1127.853,-6.135,-49.773,179.582,6.214,149.246
C03564=1127.849,-5.920,-49.785,179.583,6.218,149.247
C03565=1127.844,-5.705,-49.796,179.584,6.221,149.247
C03566=1127.840,-5.490,-49.807,179.585,6.226,149.248
C03567=1127.834,-5.240,-49.820,179.585,6.230,149.249
C03568=1127.830,-4.990,-49.833,179.585,6.234,149.250
C03569=1127.825,-4.741,-49.846,179.586,6.239,149.250
C03570=1127.819,-4.491,-49.859,179.587,6.243,149.251
C03571=1127.814,-4.241,-49.872,179.587,6.248,149.252
C03572=1127.809,-3.992,-49.884,179.588,6.253,149.253
C03573=1127.803,-3.742,-49.898,179.589,6.257,149.254
C03574=1127.799,-3.492,-49.911,179.589,6.262,149.255
C03575=1127.794,-3.243,-49.923,179.590,6.266,149.255
C03576=1127.788,-2.993,-49.936,179.591,6.271,149.256
C03577=1127.783,-2.743,-49.949,179.591,6.275,149.257
C03578=1127.778,-2.494,-49.962,179.591,6.280,149.258
C03579=1127.772,-2.244,-49.975,179.592,6.284,149.259
C03580=1127.768,-1.994,-49.988,179.593,6.289,149.259
C03581=1127.763,-1.745,-50.001,179.593,6.293,149.260
C03582=1127.757,-1.495,-50.014,179.594,6.298,149.261
C03583=1127.753,-1.246,-50.028,179.595,6.303,149.262
C03584=1127.747,-0.996,-50.041,179.595,6.306,149.263
C03585=1127.742,-0.747,-50.053,179.595,6.311,149.264
C03586=1127.737,-0.497,-50.066,179.596,6.316,149.264
C03587=1127.731,-0.247,-50.079,179.597,6.320,149.265
C03588=1127.726,0.002,-50.092,179.597,6.325,149.266
C03589=1127.721,0.252,-50.106,179.598,6.330,149.267
C03590=1127.716,0.501,-50.119,179.598,6.333,149.268
C03591=1127.711,0.751,-50.133,179.599,6.338,149.268
C03592=1127.706,1.001,-50.145,179.599,6.343,149.269
C03593=1127.700,1.250,-50.159,179.600,6.347,149.270
C03594=1127.696,1.500,-50.172,179.601,6.352,149.271
C03595=1127.691,1.749,-50.185,179.601,6.356,149.272
C03596=1127.685,1.999,-50.198,179.601,6.360,149.273
C03597=1127.680,2.248,-50.211,179.602,6.365,149.273
C03598=1127.675,2.498,-50.225,179.602,6.370,149.274
C03599=1127.670,2.748,-50.238,179.603,6.375,149.275
C03600=1127.664,2.997,-50.251,179.604,6.379,149.276
C03601=1127.660,3.247,-50.265,179.604,6.383,149.277
C03602=1127.654,3.496,-50.278,179.604,6.388,149.278
C03603=1127.650,3.746,-50.291,179.605,6.392,149.279
C03604=1127.644,3.995,-50.305,179.605,6.397,149.279
C03605=1127.639,4.245,-50.318,179.605,6.401,149.280
C03606=1127.634,4.495,-50.331,179.606,6.405,149.281
C03607=1127.629,4.745,-50.345,179.607,6.410,149.282
C03608=1127.624,4.994,-50.358,179.607,6.415,149.283
C03609=1127.618,5.244,-50.371,179.607,6.419,149.284
C03610=1127.613,5.493,-50.385,179.608,6.423,149.284
C03611=1127.608,5.743,-50.398,179.608,6.428,149.285
C03612=1127.603,5.992,-50.411,179.609,6.433,149.286
C03613=1127.598,6.242,-50.425,179.609,6.437,149.287
C03614=1127.592,6.492,-50.438,179.609,6.441,149.288
C03615=1127.588,6.707,-50.450,179.610,6.445,149.289
C03616=1127.584,6.923,-50.462,179.611,6.449,149.289
C03617=1127.580,7.138,-50.473,179.611,6.453,149.290
C03618=1127.575,7.352,-50.485,179.611,6.457,149.291
C03619=1127.571,7.568,-50.496,179.611,6.461,149.292
C03620=1127.566,7.784,-50.508,179.612,6.465,149.292
C03621=1127.561,7.999,-50.519,179.613,6.469,149.293
C03622=1127.557,8.214,-50.531,179.613,6.473,149.294
C03623=1127.552,8.464,-50.545,179.614,6.477,149.295
C03624=1127.547,8.714,-50.558,179.614,6.482,149.295
C03625=1127.542,8.963,-50.572,179.615,6.487,149.296
C03626=1127.536,9.213,-50.585,179.616,6.491,149.297
C03627=1127.532,9.462,-50.599,179.617,6.496,149.298
C03628=1127.526,9.712,-50.612,179.617,6.501,149.299
C03629=1127.521,9.962,-50.627,179.619,6.506,149.299
C03630=1127.516,10.211,-50.639,179.620,6.511,149.300
C03631=1127.511,10.461,-50.654,179.621,6.515,149.301
C03632=1127.506,10.710,-50.667,179.621,6.520,149.302
C03633=1127.501,10.960,-50.680,179.622,6.524,149.302
C03634=1127.496,11.209,-50.695,179.623,6.530,149.303
C03635=1127.490,11.459,-50.708,179.624,6.534,149.304
C03636=1127.485,11.709,-50.722,179.625,6.539,149.305
